(*
Nazwa:			FB_Robot2Bottles
Opis:			Robot podwójny
Wersja:			v0.91
Data:			2025-09-04
Autor:			TW,DP
Urzadzenia:		Mistsubishi
Konfiguracja:	
Zmiany:
- 20250904 [DP] EventLog-do sprawdzenia, 1 spr->wywołać błędy 
- 20241129 [DP] ReadyPlace w aborted, bRunProgramRC Aborted->Manual
Info: 

*)
FUNCTION_BLOCK FB_Robot2Bottles
VAR_INPUT
	bEnable									: BOOL;
	bRun									: BOOL;
	bPlace									: BOOL;
	bEStop									: BOOL;
	bHoming									: BOOL;
	bReset									: BOOL;
	iPickNumber								: INT;
	iPlaceNumber							: INT;
	bInkJetEnable							: BOOL;
	bPickOnlyOne							: BOOL; {warning 'Dorobić opcje pobierania tylko jednego opakowania, jeżeli będzie taka potrzeba'}
	iSpeed									: INT;
	iPickOffsetX							: INT;
	iPickOffsetY							: INT;  
	iPickOffsetZ							: INT; 
	iPick2OffsetX							: INT;
	iPick2OffsetY							: INT;  
	iPick2OffsetZ							: INT; 
	iPlace1OffsetX							: INT;
	iPlace1OffsetY							: INT;  
	iPlace1OffsetZ							: INT;
	iPlace2OffsetX							: INT;
	iPlace2OffsetY							: INT;
	iPlace2OffsetZ							: INT; 
	bEditOffset								: BOOL;		
	bManualMovement							: BOOL;
	iStationIndex							: UDINT;					
	sStationName							: STRING;		
	aDataRobotIOIn							: ARRAY[1..8] OF USINT;
	aDataRobotREGIn							: ARRAY[1..32] OF UINT;
	
	iCaseReset								: INT;
	
	iAxisId									: INT;	
	bBatteryReplacementWasMade				: BOOL;
	bGreaseReplacementWasMade				: BOOL;
	bBeltReplacementWasMade					: BOOL;
	bWarningAcknowledge						: BOOL;




END_VAR

VAR_OUTPUT
	
	eState									: E_Station;						//Stan ogólny bloku
	eRunningState							: E_RobotMovState;					//Stan podbloku
	bError									: BOOL;								//Błąd stacji
	udiErrorId								: UDINT;							//Nr błędu grzałki zasadniczej
	sErrorDescription1						: STRING(200);							//Opis błędu
	sErrorDescription2						: STRING(200);							//Opis błędu
	sErrorStationName						: STRING;							//Nazwa stacji
	udiStationID							: UDINT;							// Nr stacji

	tCycleTime								: TIME;	
	bHomingDone								: BOOL;								//Bazowanie wykonane
	bHomingNeeded 							: BOOL;								
	bCycleDone								: BOOL;
	bCycleNotDone							: BOOL;
	iLastPickNumber							: INT;
	iBottleTransferLock						: INT;
	aActualPosition							: ARRAY[0..3] OF INT;
	aLoadAxis								: ARRAY[0..3] OF INT;
	aDataRobotIOOut							: ARRAY[1..8] OF USINT;
	aDataRobotREGOut						: ARRAY[1..32] OF UINT;
	bWarning								: BOOL;
	sWarningDescription1					: STRING;
	sWarningDescription2					: STRING;
	udiWarningId							: UDINT;
	
	
END_VAR

VAR_IN_OUT
	
	bManualPick								: BOOL;
	bManualPick2							: BOOL;
	bManualPlace1							: BOOL;
	bManualPlace2							: BOOL;
	bManualReadyPosition					: BOOL;
	bManualStartInkJetPosition				: BOOL;
	bManualStopInkJetPosition				: BOOL;
	bManualWeightPosition					: BOOL;
	bManualCatch							: BOOL;
	nLubricationCounter						: DINT;	//Licznik czasu samrowania
END_VAR

VAR
	iCaseRC									: INT;
	iLastCaseRC								: INT;
	iActualCase								: INT;	
	iCaseInit								: INT;
	iCaseHoming								: INT;
	iCaseManual								: INT;
	iTemperatureRC							: INT;
	bReadyRC								: BOOL;
	bSafePositionRC							: BOOL;
	bResetErrorRC							: BOOL;
	bErrorRCActive							: BOOL;
	bServoONRC								: BOOL;
	bServoONRCActive						: BOOL;
	bServoOFFRC								: BOOL;
	bServoOFFRCActive						: BOOL;
	bOperationEnableRC						: BOOL;
	bOperationEnableRCActive				: BOOL;
	bErrorNumberRequest						: BOOL;
	bRunProgramRC							: BOOL;
	bRunProgramRCActive						: BOOL;
	bProgramResetRC							: BOOL;
	bProgramSelectRCActive					: BOOL;
	bCatcherCloseSensor						: BOOL;
	bComingUp								: BOOL;
	bSlowMotion								: BOOL;
	IODATA									: UDINT;
	ftCapFeederRobotEditOffset				: F_TRIG;
	rtCapFeederRobotEditOffset				: R_TRIG;
	tonRetryInit							: TON;	
	tonErrorDelay							: TON;	
	tonReadyError							: TON;
	iErrorCase								: INT;
	iSpeedSend								: INT;

	tonWaitForSuckerSensor					: TON;
	iZ										: INT;
	rtPick									: R_TRIG;
	
	iActualLastCase							: INT;
	aDataRobotIn							: INT;
	rtrigCycleTimerRead						: R_TRIG;
	tonCycleTimer							: TON;
	bLowLevelErrorRCActive					: BOOL;
	bWarningRCActive						: BOOL;
	bBatteryLowVoltage						: BOOL;
	bBatteryReplenishmentFinished			: BOOL;
	bGreaseReplenishmentFinished			: BOOL;
	bBeltReplenishmentFinished				: BOOL;
	tonbStateError							: TON;
	bStateError								: BOOL;
	udiHighLevelErrorId						: UDINT;
	udiMaintenanceErrorId					: UDINT;
	udiLowLevelErrorId						: UDINT;
	rtPlace									: R_TRIG;
	bHighLevelErrorRCActive					: BOOL;
	bErrorNumberRequestActive				: BOOL;
	
	fbIntTo2Byte							: FB_IntTo2Byte;
	IODATATest								: UDINT;
// dane wysyłane liczbowo do robota	
	udiIoDATARCWrite						: UDINT;	
	
	
// Wymiana smaru i paskow	
// Sygnaly wystawiane do robota
	bBatteryReplacementDone			: BOOL;	
	bGreaseReplacementDone			: BOOL;	
	bBeltReplacementDone			: BOOL;	

	
	bBeltReplacementDoneAxis3		: BOOL;
	bBeltReplacementDoneAxis4		: BOOL;
	
	bGreaseReplacementDoneAxis1		: BOOL;	
	bGreaseReplacementDoneAxis2		: BOOL;	
	bGreaseReplacementDoneAxis3		: BOOL;	
	
	
	udiErrorIdInit: UDINT;
	bWarningNumberRequest: BOOL;

	bResetWarningRC: BOOL;
	
	
		//Zmienne od EVENTLOGGER
	bAlarmInit 						: BOOL := TRUE; 
	nAlarmNumerator					: INT;
	arfbAlarm						: ARRAY[0..19] OF  FB_TcAlarm;		//Tablica bloczków błędów
	fbSourceInfo 					: FB_TcSourceInfo;
	iSourceInfo						: I_TcSourceInfo;
	sAlarmTest						: STRING;
	//Koniec zmiennych od EVENTLOGGER
END_VAR


Control();
DataExchange();
ErrorHandling();
Warning();
LubricationCounter();
aStatistic();
aStationID();

//Zabezpieczneie przed błędem 0 dp
IF udiErrorId = 0 AND bError THEN
	udiErrorId := 311;
	//udiErrorId := 999;	
END_IF

ACTION aStationID:
udiStationID	:=	iStationIndex;
END_ACTION

ACTION aStatistic:

//Statystyka do zliczania czasu cyklu 
rtrigCycleTimerRead(CLK:=bCycleDone);


	IF rtrigCycleTimerRead.Q THEN
		tCycleTime:=tonCycleTimer.ET;
	END_IF
	
tonCycleTimer(IN:= eRunningState<>E_RobotMovState.eReadyPlace , PT:=T#1D);
END_ACTION

ACTION Control:

	iSpeedSend := iSpeed;
	
	IF iPlaceNumber = 2 THEN
		iSpeedSend := REAL_TO_INT(iSpeed / 2);
	END_IF
	
	(*****Wyłączenie enable*****)
	IF NOT bEnable THEN
		IF eState <> E_Station.eDisabled AND eState <> E_Station.ePreparingToDisable THEN
				eState 				:= E_Station.ePreparingToDisable; 
		END_IF	
	END_IF

	(*****Estop*****)
	IF NOT bEstop  THEN	
		IF eState <> E_Station.eAborted AND eState <> E_Station.eAborting AND eState <> E_Station.eDisabled THEN
				eState 				:= E_Station.eAborting; 
		END_IF
	END_IF

	
	CASE eState OF
	/////////////////////////////	
		E_Station.eDisabled: 					// Stan nieaktywnosci (Stacja wyłączona) 
		
			iCaseInit				:= 0;
			IF bEnable THEN
				eState 				:= E_Station.ePreparingToReady; 
			END_IF 
			
    /////////////////////////////	    
		E_Station.eAborted: 					// Stan bezpiecznego zatrzymania (po Abortingu) 
			
			bServoONRC							:= FALSE;
			bRunProgramRC						:= FALSE;
			bResetErrorRC						:= FALSE;		
			IF bEStop THEN
				eState 				:= E_Station.ePreparingToReady;
				iCaseInit			:=0;
				eRunningState		:=	E_RobotMovState.eReadyPlace;	
			//iActualCase			:= iActualLastCase;
				//IF iActualLastCase = 200 THEN
				//	iActualCase := 250;
				//END_IF
			END_IF
			
	/////////////////////////////	
		E_Station.eAborting:                 	// Stan bezpiecznego zatrzymywania (po EStopie)
			eState 					:=	E_Station.eAborted;  
			iActualLastCase			:=	iActualCase;
		
			
	/////////////////////////////			
		E_Station.eError:                 	 	// Stan błędu 	
	
			iCaseInit				:= 0;
			//bServoONRC			:= FALSE;
			bManualPick			:= FALSE;
			bManualPick2			:= FALSE;
			bManualPlace1				:= FALSE;
			bManualPlace2					:= FALSE;
			
			IF bReset THEN
				eState 				:= E_Station.eResetting;
			END_IF
			
			IF NOT bError THEN
				eState 				:=	E_Station.ePreparingToReady;
				iCaseInit			:=0;
			END_IF
			
	/////////////////////////////
		E_Station.eResetting:					// Stan resetowania bledu (po Errorze)
			
			IF bError THEN
				
				bResetErrorRC					:= bReset;
				eRunningState					:= E_RobotMovState.eReadyPlace;
				bHomingDone						:= FALSE;
				udiErrorId						:= 0;
			END_IF
				
			IF NOT bErrorRCActive  THEN
				bError							:= FALSE;
				bResetErrorRC					:= FALSE;
				bErrorNumberRequest				:= FALSE;				
			END_IF
			
			IF NOT bError THEN
				udiErrorId 			:=	0;
   				sErrorDescription1 	:=	'';
   				sErrorDescription2 	:=	'';				
				eState 				:=	E_Station.ePreparingToReady;
				eRunningState		:=	E_RobotMovState.eReadyPlace;
				iCaseInit			:=0;
//			ELSE
//				eState 				:=	E_Station.eError;
			END_IF
        
	/////////////////////////////
		E_Station.eManualMovement:     			// Stan ruchów manualnych  
       
			ManualMovements();
			//Wyjście z trybu serwisowego
			IF NOT bManualMovement THEN
				eState:=E_Station.eReady;
			END_IF
			IF bHoming THEN
				iCaseHoming					:= 0;
				eState 						:= E_Station.eHoming; 
			END_IF

	/////////////////////////////
		E_Station.eHoming:						// Stan bazowania 
	
			Homing();
			IF NOT bHoming THEN
			   eState:=E_Station.ePreparingToReady;
			   iCaseInit			:=0;
			END_IF		
			
	/////////////////////////////
		E_Station.eHomingDone:                  // Stan wykonania bazowania 
		
			iZ:=iZ+1;
			IF NOT bHoming THEN
			   eState:=E_Station.eReady;
			END_IF
			
	/////////////////////////////
		E_Station.ePreparingToReady:            // Stan przygotowywania do gotowosci (zawsze przed Ready)  
			iCaseRC								:= 0;
			Init();
			
			
	/////////////////////////////
		E_Station.ePreparingToDisable:          // Stan przygotowywania do nieaktywnosci (po wyłączeniu Enable) 
  	
				eState:=E_Station.eDisabled;
			
	/////////////////////////////
		E_Station.eReady:						// Stan gotowosci 
		
			bServoONRC							:= TRUE;
			
			IF bServoONRCActive THEN
				bRunProgramRC					:= TRUE;			
			END_IF
		
			IF bRun AND NOT bCycleDone AND NOT bCycleNotDone THEN
				eState 						:= E_Station.eStarting; 
			END_IF
			
			
			IF bManualMovement AND bRunProgramRC THEN
				//Jeśli przejście w tryb ruchów manualnych przepisz wszystkie stany siłowników sterowanych przez moduł
				//aby zapobiec ewentualnym kolizjom po wejściu w tryb serwisowy
				iCaseManual					:= 0;
				eState 						:= E_Station.eManualMovement; 
			END_IF
			
			IF NOT bRun THEN
				bCycleDone 					:= FALSE;
				bCycleNotDone 				:= FALSE;			
			END_IF
			
			
			IF bHoming THEN
				iCaseHoming					:= 0;
				eState 						:= E_Station.eHoming; 
			END_IF
			
			
			iCaseRC							:= 0;			//22.07.2020
			
			//eRunningState					:=	E_RobotMovState.eReadyPlace;
			
			
		
			
	/////////////////////////////
		E_Station.eStopping:					// Stan zatrzymywania 

			eState 							:= E_Station.eReady;	
			
	/////////////////////////////
		E_Station.eStarting:                  	// Stan uruchamiania (po Ready)	
			bResetErrorRC					:= FALSE;	
			eState					 		:= E_Station.eRunning; 
			
	/////////////////////////////
		E_Station.eRunning:               		// Stan wykonywania cyklu (po Startingu), w tym stanie osobny
 

			IF NOT bRun AND NOT bCycleDone THEN					(*Przerywanie cyklu*)
				eState 				 		:= E_Station.eStopping;	
			END_IF
			
			IF bCycleDone OR bCycleNotDone THEN (*Cykl zakończony*)
				eState 				 		:= E_Station.eReady;
				eRunningState						:=	E_RobotMovState.eReadyPlace;
			END_IF		
			
			Running();
			
			
	/////////////////////////////		
	END_CASE
END_ACTION

ACTION DataExchange:


//SignalOutput
aDataRobotIOOut[1].0                	:= bOperationEnableRC;
aDataRobotIOOut[1].1                	:= bRunProgramRC;
aDataRobotIOOut[1].2              		:= bSlowMotion;
aDataRobotIOOut[1].3                	:= bProgramResetRC;
aDataRobotIOOut[1].4                	:= bServoONRC;
aDataRobotIOOut[1].5                	:= bServoOFFRC;
aDataRobotIOOut[1].6                	:= bResetErrorRC OR bResetWarningRC;
aDataRobotIOOut[1].7                	:= bEditOffset;
aDataRobotIOOut[2].0                	:= bManualCatch;
aDataRobotIOOut[2].1                	:= bErrorNumberRequest OR bWarningNumberRequest;
//Dodane Darek
aDataRobotIOOut[2].7                	:= bBatteryReplacementDone;		//6015
aDataRobotIOOut[3].0                	:= bGreaseReplacementDone;		//6016
aDataRobotIOOut[3].1                	:= bBeltReplacementDone;		//6017
aDataRobotIOOut[3].2                	:= bBeltReplacementDone;		//6017

//SignalRegOutput
aDataRobotREGOut[1]                    	:= INT_TO_UINT(iCaseRC);
aDataRobotREGOut[2]                    	:= INT_TO_UINT(iSpeedSend);
aDataRobotREGOut[3]                    	:= INT_TO_UINT(iPickOffsetX);
aDataRobotREGOut[4]                    	:= INT_TO_UINT(iPickOffsetY);
aDataRobotREGOut[5]                    	:= INT_TO_UINT(iPickOffsetZ);
aDataRobotREGOut[6]                    	:= INT_TO_UINT(iPlace1OffsetX);
aDataRobotREGOut[7]                  	:= INT_TO_UINT(iPlace1OffsetY);
aDataRobotREGOut[8]                    	:= INT_TO_UINT(iPlace1OffsetZ);
aDataRobotREGOut[9]                    	:= INT_TO_UINT(iPlace2OffsetX);
aDataRobotREGOut[10]                	:= INT_TO_UINT(iPlace2OffsetY);
aDataRobotREGOut[11]                	:= INT_TO_UINT(iPlace2OffsetZ);
//Dodane Darek
aDataRobotREGOut[12]                    := INT_TO_UINT(iPick2OffsetX);
aDataRobotREGOut[13]                    := INT_TO_UINT(iPick2OffsetY);
aDataRobotREGOut[14]                    := INT_TO_UINT(iPick2OffsetZ);

// IODATA

fbIntTo2Byte(
iInput:= UDINT_TO_INT(udiIoDATARCWrite), 
byStarszy=> , 
byMlodszy=> );


aDataRobotIOOut[8]												:= fbIntTo2Byte.byStarszy;
aDataRobotIOOut[7]												:= fbIntTo2Byte.byMlodszy;

// Testowy odczyt wartosci wysyłanej
IODATATest                                	:= WORD_TO_UDINT(F_2Bytes_To_Word(aDataRobotIOOut[8], aDataRobotIOOut[7]));


//SignalInput                               
bOperationEnableRCActive            	:= aDataRobotIOIn[1].0;		//6000
bRunProgramRCActive                   	:= aDataRobotIOIn[1].1;
//                                    	:= aDataRobotIOIn[1].2;
bProgramSelectRCActive                	:= aDataRobotIOIn[1].3;
bServoONRCActive                    	:= aDataRobotIOIn[1].4;
bServoOFFRCActive                    	:= aDataRobotIOIn[1].5;
bErrorRCActive                        	:= aDataRobotIOIn[1].6;
bReadyRC                            	:= aDataRobotIOIn[1].7;
bSafePositionRC                        	:= aDataRobotIOIn[2].0;		//6008
bErrorNumberRequestActive               := aDataRobotIOIn[2].1;
bCatcherCloseSensor                    	:= aDataRobotIOIn[2].2;

//Dodane Darek
bHighLevelErrorRCActive                 := aDataRobotIOIn[2].3;		//6011
bLowLevelErrorRCActive                  := aDataRobotIOIn[2].4;		//6012
bWarningRCActive                    	:= aDataRobotIOIn[2].5;		//6013
bBatteryLowVoltage              		:= aDataRobotIOIn[2].6;		//6014
bBatteryReplenishmentFinished               := aDataRobotIOIn[2].7;		//6015
bGreaseReplenishmentFinished	            := aDataRobotIOIn[3].0;		//6016
bBeltReplenishmentFinished	                := aDataRobotIOIn[3].1;		//6017



//SignalRegInput
iActualCase                            	:= UINT_TO_INT(aDataRobotREGIn[1]);
aLoadAxis[0]                        	:= UINT_TO_INT(aDataRobotREGIn[2]);
aLoadAxis[1]                        	:= UINT_TO_INT(aDataRobotREGIn[3]);       
aLoadAxis[2]                        	:= UINT_TO_INT(aDataRobotREGIn[4]);       
aLoadAxis[3]                        	:= UINT_TO_INT(aDataRobotREGIn[5]);
IODATA                                	:= WORD_TO_UDINT(F_2Bytes_To_Word(aDataRobotIOIn[8], aDataRobotIOIn[7]));
END_ACTION

ACTION ErrorDescription:
IF bErrorRCActive AND bHighLevelErrorRCActive THEN

		CASE udiHighLevelErrorId OF	
			
			
0001:					
					
	sErrorDescription1 := 'Fail safe error (SRVOFF).  System problem.';				
	sErrorDescription2 := 'Turn the power OFF and ON once. When it comes back, contact to the dealer.';				
					
0002:					
					
	sErrorDescription1 := 'Fail safe error (STOP).  System Problem.';				
	sErrorDescription2 := 'Turn the power OFF and ON once. When it comes back, contact to the dealer.';				
					
0003:					
					
	sErrorDescription1 := 'System fail.  System Problem.';				
	sErrorDescription2 := 'Check System.When it comes back, contact to the dealer.';				
					
0004:					
					
	sErrorDescription1 := 'CPU Watch dog error.  CPU was not normally treatable.';				
	sErrorDescription2 := 'It is necessary to change some parts when not improvement';				
					
0005:					
					
	sErrorDescription1 := 'Turn the power OFF and ON onc.  The robot model was selected..';				
	sErrorDescription2 := 'Turn the power OFF and ON once';				
					
0006:					
					
	sErrorDescription1 := ' CPU process error.  CPU was not normally treatable.';				
	sErrorDescription2 := 'It is necessary to change some parts when not improvement';				
					
0008:					
					
	sErrorDescription1 := ' CPU synchronization error.  CPU synchronization was failed.';				
	sErrorDescription2 := 'Turn the power OFF and ON once';				
					
0009:					
					
	sErrorDescription1 := 'Version UP (ALL).  Version UP (ALL).';				
	sErrorDescription2 := 'Turn the power OFF,ROTSW=0 and power ON once';				
					
0010:					
					
	sErrorDescription1 := 'Illeagal Version (file).  Version is different.';				
	sErrorDescription2 := 'File was initialized';				
					
0011:					
					
	sErrorDescription1 := 'Illeagal Version (system data.  Version is different.';				
	sErrorDescription2 := 'System data was initialized';				
					
0012:					
					
	sErrorDescription1 := 'Initialize (error log).  Version is different or illegal log file.';				
	sErrorDescription2 := 'Error log was initialized';				
					
0014:					
					
	sErrorDescription1 := 'System error (illegal MECHA).  System error (illegal MECHA).';				
	sErrorDescription2 := 'Set the correct MECHA';				
					
0015:					
					
	sErrorDescription1 := 'Illeagal Version (file).  System ERROR 1.';				
	sErrorDescription2 := 'Contact the maker.';				
					
0016:					
					
	sErrorDescription1 := 'Turn the power OFF and ON onc.  Power OFF/ON a little more slowly,please.';				
	sErrorDescription2 := 'Turn the power OFF and ON once';				
					
0017:					
					
	sErrorDescription1 := '  EEPROM error.  EEPROM is broken.';				
	sErrorDescription2 := 'It is necessary to replace the CPU board';				
					
0019:					
					
	sErrorDescription1 := 'Illegal RotSW on CPU.  RotSW is set not 0.';				
	sErrorDescription2 := 'Please set RotSW to 0';				
					
0020:					
					
	sErrorDescription1 := 'System Error(same name is Bac.  System Error(same name is Backup data.).';				
	sErrorDescription2 := 'Change the system software';				
					
0021:					
					
	sErrorDescription1 := 'System Error(Backup data is C.  System Error(Backup data is Count over.).';				
	sErrorDescription2 := 'Change the system software';				
					
0022:					
					
	sErrorDescription1 := 'System Error(Backup data is n.  System Error(Backup data is no area.).';				
	sErrorDescription2 := 'Change the system software';				
					
0025:					
					
	sErrorDescription1 := ' Files will be saved to ROM.  Program and parameter files will be saved to ROM.';				
	sErrorDescription2 := 'Turn the power OFF and power ON once';				
					
0026:					
					
	sErrorDescription1 := ' Files will be loaded from ROM.  Program and parameter files will be loaded from ROM.';				
	sErrorDescription2 := 'Turn the power OFF and power ON once';				
					
0027:					
					
	sErrorDescription1 := ' Backup or restore is canceled.  Backup or restore is canceled.';				
	sErrorDescription2 := 'Turn the power OFF and power ON once';				
					
0028:					
					
	sErrorDescription1 := ' Memory error (ECC).  2bit error of ECC was detected.';				
	sErrorDescription2 := 'Turn the power OFF and ON once';				
					
0039:					
					
	sErrorDescription1 := 'Door Switch Signal line is fa.  Door Switch Signal line is faulty..';				
	sErrorDescription2 := 'Check the Door Switch Signal line';				
					
0040:					
					
	sErrorDescription1 := 'Door Switch Signal is Input.  Door Switch is opened.';				
	sErrorDescription2 := 'Please close the Door be connected with Door Switch';				
					
0041:					
					
	sErrorDescription1 := 'Comm. error (Remote I/O #1).  Communication line is illegal.';				
	sErrorDescription2 := 'Check the cable or power supply';				
					
0042:					
					
	sErrorDescription1 := ' Comm. error (Remote I/O #2).  Communication line is illegal.';				
	sErrorDescription2 := 'Check the cable or power supply';				
					
0043:					
					
	sErrorDescription1 := ' Comm. error (Remote I/O #3).  Communication line is illegal.';				
	sErrorDescription2 := 'Check the cable or power supply';				
					
0044:					
					
	sErrorDescription1 := ' Comm. error (Remote I/O #4).  Communication line is illegal.';				
	sErrorDescription2 := 'Check the cable or power supply';				
					
0045:					
					
	sErrorDescription1 := ' Comm. error (Remote I/O #5).  Communication line is illegal.';				
	sErrorDescription2 := 'Check the cable or power supply';				
					
0046:					
					
	sErrorDescription1 := ' Faulty wiring (Mode sel. swit.  The state of doubled wiring is not matching (Mode sel. switch).';				
	sErrorDescription2 := 'Please check the wiring (Mode sel. switch)';				
					
0047:					
					
	sErrorDescription1 := ' OCL detect.  OCL detect.';				
	sErrorDescription2 := 'Please check the line (O/P Emergency Stop)';				
					
0048:					
					
	sErrorDescription1 := ' Faulty line (Mode Selector SW.  The state of doubled line is not matching (Mode Selector switch).';				
	sErrorDescription2 := 'Please check the line (Mode Selector switch)';				
					
0049:					
					
	sErrorDescription1 := ' Faulty Line (T/B Enable Switc.  The state of doubled line is not matching (T/B Enable Switch).';				
	sErrorDescription2 := 'Please check the line (T/B Enable Switch)';				
					
0050:					
					
	sErrorDescription1 := 'EMG signal is input. (externa.  EMG signal is input. (external).';				
	sErrorDescription2 := 'Check the external emergency stop';				
					
0051:					
					
	sErrorDescription1 := 'EMG line is faulty.(external).  EMG line is faulty.(external).';				
	sErrorDescription2 := 'Check the external emergency stop';				
					
0052:					
					
	sErrorDescription1 := ' EMG signal is input.(Add.Axis.  EMG signal is input.(Add.Axis1).';				
	sErrorDescription2 := 'Check the emergency stop of Additional Axis card';				
					
0053:					
					
	sErrorDescription1 := 'EMG signal is input.(Add.Axis.  EMG signal is input.(Add.Axis).';				
	sErrorDescription2 := 'Check the emergency stop of Additional Axis servo amp.';				
					
0054:					
					
	sErrorDescription1 := ' Faulty wiring (External EMG p.  The state of doubled wiring is not matching (External EMG).';				
	sErrorDescription2 := 'Please check the wiring (External Emergency Stop)';				
					
0060:					
					
	sErrorDescription1 := 'EMG signal is input. (O.Panel.  EMG signal is input. (O.Panel).';				
	sErrorDescription2 := 'Check the O.Panel emergency stop';				
					
0061:					
					
	sErrorDescription1 := 'EMG line is faulty.(0.Panel).  EMG line is faulty.(0.Panel).';				
	sErrorDescription2 := 'Check the O.Panel emergency stop';				
					
0070:					
					
	sErrorDescription1 := 'EMG signal is input. (T.Box).  EMG signal is input. (T.Box).';				
	sErrorDescription2 := 'Check the T.Box emergency stop';				
					
0071:					
					
	sErrorDescription1 := 'EMG line is faulty.(T.Box).  EMG line is faulty.(T.Box).';				
	sErrorDescription2 := 'Check the T.Box emergency stop';				
					
0072:					
					
	sErrorDescription1 := 'EMG cancel operation is fault.  TB cancel switch operation was incorrect.';				
	sErrorDescription2 := 'Check the T/B cancel switch operation';				
					
0073:					
					
	sErrorDescription1 := 'EMG cancel line is faulty.(T..  EMG cancel line is faulty.(T.Box).';				
	sErrorDescription2 := 'Check the EMG cancel line';				
					
0074:					
					
	sErrorDescription1 := 'Faulty line (T/B Enable/Disab.  The state of doubled line is not matching (T/B Enable/Disable).';				
	sErrorDescription2 := 'Please check the line (T/B Enable/Disable)';				
					
0075:					
					
	sErrorDescription1 := 'TB communication error.  Communication between the RC and TB was cut off.';				
	sErrorDescription2 := 'Check TB communication line';				
					
0076:					
					
	sErrorDescription1 := 'TB connection error.  Cannot detect TB connection.';				
	sErrorDescription2 := 'If this error recurs, please contact us';				
					
0077:					
					
	sErrorDescription1 := ' Electric double layer overvol.  A power supply of a substrate in the robot is broken.';				
	sErrorDescription2 := 'Turn the power OFF and contact your service provider';				
					
0079:					
					
	sErrorDescription1 := ' Contactor of converter unit e.  Contactor of converter unit is closed.';				
	sErrorDescription2 := 'Confirm status of contactor of converter unit';				
					
0080:					
					
	sErrorDescription1 := ' Fuse of brake line is blown.  Fuse of brake line is blown.';				
	sErrorDescription2 := 'Change fuse';				
					
0081:					
					
	sErrorDescription1 := ' Fuse is blown.(motor hand I/F.  Fuse is blown.(motor hand I/F).';				
	sErrorDescription2 := 'Change fuse';				
					
0082:					
					
	sErrorDescription1 := 'Fuse is broken (air hand I/F).  Fuse is blown.(air hand I/F).';				
	sErrorDescription2 := 'Change fuse';				
					
0083:					
					
	sErrorDescription1 := 'Fuse is broken(hand input pow.  Fuse is blown.(hand input power).';				
	sErrorDescription2 := 'Change fuse';				
					
0084:					
					
	sErrorDescription1 := 'Fuse is broken(O/P).  Fuse is blown.(O/P).';				
	sErrorDescription2 := 'Change fuse';				
					
0085:					
					
	sErrorDescription1 := ' Fuse is blown.(External EMG).  Open phase in the input power.';				
	sErrorDescription2 := 'Change fuse';				
					
0086:					
					
	sErrorDescription1 := 'Hand module overcurrent.  Hand module is broken.';				
	sErrorDescription2 := 'Change Hand module';				
					
0087:					
					
	sErrorDescription1 := 'Fuse is blown.(Brake).  Fuse is blown.(Brake).';				
	sErrorDescription2 := 'Change fuse';				
					
0088:					
					
	sErrorDescription1 := ' Fuse is blown.(Service I/F).  Fuse is blown.(Service I/F).';				
	sErrorDescription2 := 'Please confirm the input and output current of service I/F. ';				
					
0089:					
					
	sErrorDescription1 := ' Fuse of external battery is b.  Fuse of external battery is blown..';				
	sErrorDescription2 := 'Check that an outside power-supply voltage is 4.5V or less.';				
					
0090:					
					
	sErrorDescription1 := ' Fuse is blown..  Fuse is blown.';				
	sErrorDescription2 := 'Change fuse';				
					
0093:					
					
	sErrorDescription1 := ' Safety relay fuse is blown..  Safety relay fuse is blown..';				
	sErrorDescription2 := 'Change fuse.';				
					
0094:					
					
	sErrorDescription1 := ' The fuse in the T/B was blown.  The fuse in the T/B power supply line was blown..';				
	sErrorDescription2 := 'Please check the earth fault of the T/B cable.';				
					
0097:					
					
	sErrorDescription1 := ' Faulty status (MC).  The state of doubled signal is not matching (MC status).';				
	sErrorDescription2 := 'Turn the power OFF and ON once';				
					
0098:					
					
	sErrorDescription1 := ' Faulty status (SR).  The state of doubled signal is not matching (SR status).';				
	sErrorDescription2 := 'Turn the power OFF and ON once';				
					
0099:					
					
	sErrorDescription1 := ' S/W with an old version is in.  S/W with an old version is installed.';				
	sErrorDescription2 := 'Install the S/W with a correct version';				
					
0100:					
					
	sErrorDescription1 := 'Temperature in the Controlle .  FAN check or Filter at the bottom on Controller becomes old.';				
	sErrorDescription2 := 'Please exchange the filter to new filter or clean up the filter';				
					
0103:					
					
	sErrorDescription1 := ' Temp. in robot CPU is too hig.  Ambient temperature of robot CPU becomes high.';				
	sErrorDescription2 := 'Please lower ambient temperature to the specification range';				
					
0117:					
					
	sErrorDescription1 := ' Power supply error (brake).  The output of the power supply deviated from the specified range.';				
	sErrorDescription2 := 'Turn the power OFF and contact your service provider';				
					
0130:					
					
	sErrorDescription1 := 'System RemoteI/O down.  Communication line of System Remote I/O is illegal.';				
	sErrorDescription2 := 'Check the cable or power supply';				
					
0131:					
					
	sErrorDescription1 := ' Plural Ope-panel are installe.  One operation panel can be installed..';				
	sErrorDescription2 := 'Install only one operation panel.';				
					
0140:					
					
	sErrorDescription1 := 'Fuse is blown.(Safety unit).  Fuse is blown.(Safety unit).';				
	sErrorDescription2 := 'Change fuse';				
					
0141:					
					
	sErrorDescription1 := ' Wiring error of EMGIN connect.  Wiring error of EMGIN connector.';				
	sErrorDescription2 := 'Please confirm the wiring for EMGIN';				
					
0160:					
					
	sErrorDescription1 := 'Cannot use PIO I/F and Unit.  The I/O Channel number of PIO interface and PIO unit overlaps..';				
	sErrorDescription2 := 'Select either of Paralle I/O interface or Paralle I/O unit.';				
					
0162:					
					
	sErrorDescription1 := 'Cannot use PIO I/F and Unit.  The I/O Channel number of PIO interface and PIO unit overlaps..';				
	sErrorDescription2 := 'Select either of Paralle I/O interface or Paralle I/O unit.';				
					
0163:					
					
	sErrorDescription1 := 'Cannot use PIO I/F and Unit.  The I/O Channel number of PIO interface and PIO unit overlaps..';				
	sErrorDescription2 := 'Select either of Paralle I/O interface or Paralle I/O unit.';				
					
0170:					
					
	sErrorDescription1 := 'Parallel I/O interface H/W er.  The card might be broken..';				
	sErrorDescription2 := 'Please exchange the Parallel I/O interface card.';				
					
0172:					
					
	sErrorDescription1 := 'Parallel I/O interface H/W er.  The card might be broken..';				
	sErrorDescription2 := 'Please exchange the Parallel I/O interface card.';				
					
0173:					
					
	sErrorDescription1 := 'Parallel I/O interface H/W er.  The card might be broken..';				
	sErrorDescription2 := 'Please exchange the Parallel I/O interface card.';				
					
0180:					
					
	sErrorDescription1 := 'Fuse is blown.(PIO) （Slot 1-F.  Fuse is blown.(Paralle I/O interface).';				
	sErrorDescription2 := 'Change fuse (Paralle I/O interface)';				
					
0182:					
					
	sErrorDescription1 := 'Fuse is blown.(PIO) （Slot 2-F.  Fuse is blown.(Paralle I/O interface).';				
	sErrorDescription2 := 'Change fuse (Paralle I/O interface)';				
					
0183:					
					
	sErrorDescription1 := 'Fuse is blown.(PIO) （Slot 3-F.  Fuse is blown.(Paralle I/O interface).';				
	sErrorDescription2 := 'Change fuse (Paralle I/O interface)';				
					
0210:					
					
	sErrorDescription1 := ' Power supply error.  The output of the power supply deviated from the specified range.';				
	sErrorDescription2 := 'Turn the power OFF and ON once';				
					
0211:					
					
	sErrorDescription1 := ' Power supply error.  The output of the power supply deviated from the specified range.';				
	sErrorDescription2 := 'Turn the power OFF and ON once';				
					
0212:					
					
	sErrorDescription1 := ' Power supply error.  The output of the power supply deviated from the specified range.';				
	sErrorDescription2 := 'Turn the power OFF and ON once';				
					
0213:					
					
	sErrorDescription1 := ' Power supply error.  The output of the power supply deviated from the specified range.';				
	sErrorDescription2 := 'Turn the power OFF and ON once';				
					
0220:					
					
	sErrorDescription1 := ' Memory error (Main CPU).  Memory error was detected (Main CPU).';				
	sErrorDescription2 := 'Turn the power OFF and ON once';				
					
0230:					
					
	sErrorDescription1 := ' Safety parameter error.  Detect errors in safety parameter value.';				
	sErrorDescription2 := 'Please check the safety parameter setting';				
					
0231:					
					
	sErrorDescription1 := ' Parameter CRC error.  Detect CRC errors in safety parameter.';				
	sErrorDescription2 := 'Please check the safety parameters settings and write parameters';				
					
0241:					
					
	sErrorDescription1 := ' Fault in Safety Communication.  Detect a fault in safety communication.';				
	sErrorDescription2 := 'Turn the power OFF and ON once';				
					
0242:					
					
	sErrorDescription1 := ' Fault in Safety Data.  Detect a fault in safety data.';				
	sErrorDescription2 := 'Turn the power OFF and ON once';				
					
0243:					
					
	sErrorDescription1 := ' Safety function unavailable.  The Safety Function is not supported by this robot.';				
	sErrorDescription2 := 'Disable the safety function';				
					
0260:					
					
	sErrorDescription1 := ' EMG circuit diagnosis error.  Voltage diagnosis error.';				
	sErrorDescription2 := 'Turn the power OFF and ON once';				
					
0270:					
					
	sErrorDescription1 := ' Voltage diagnosis error.  Voltage diagnosis error.';				
	sErrorDescription2 := 'Turn the power OFF and ON once';				
					
0280:					
					
	sErrorDescription1 := ' STO circuit diagnosis error.  STO citcuit error.';				
	sErrorDescription2 := 'Turn the power OFF and ON once';				
					
0290:					
					
	sErrorDescription1 := ' PLD control error.  PLD control error.';				
	sErrorDescription2 := 'Turn the power OFF and ON once';				
					
0300:					
					
	sErrorDescription1 := ' CR800 test H-Error.  General-purpose H-Error for the function test of CR800.';				
	sErrorDescription2 := 'Check the embedded message';				
					
0310:					
					
	sErrorDescription1 := ' Mecha board access error.  Failed in access to a Mecha board.';				
	sErrorDescription2 := 'Please confirm the connection with Mecha board';				
					
0311:					
					
	sErrorDescription1 := ' RemoteI/O unit config error.  The multiple RemoteI/O units which do not support are connected.';				
	sErrorDescription2 := 'Please confirm the constitution of RemoteI/O unit';				
					
0315:					
					
	sErrorDescription1 := ' Can not access the D-device are.  This area cannot be used in duplicate.';				
	sErrorDescription2 := 'Please change the D-device start number in parameter DDEVVLn';				
					
0316:					
					
	sErrorDescription1 := ' The D-device area is out of r.  An area corresponding to the variable type can not be allocated.';				
	sErrorDescription2 := 'Please change the D-device start number in parameter DDEVVLn';				
					
0317:					
					
	sErrorDescription1 := ' The D-device variable duplica.  Cannot be doubly allotted to one variable.';				
	sErrorDescription2 := 'Please change the variable name in parameter DDEVVLn';				
					
0470:					
					
	sErrorDescription1 := ' Abnormality of DB(Add.Axis).  The addition axis dynamic brake is abnormal.';				
	sErrorDescription2 := 'Check the dynamic brake unit and the cable connection';				
					
0490:					
					
	sErrorDescription1 := 'Alarm of fan in the robot.  Fan in the robot might be out of order.';				
	sErrorDescription2 := 'Please exchange the fan in the robot';				
					
0491:					
					
	sErrorDescription1 := 'Alarm of fan1 in the robot.  Fan1 in the robot might be out of order.';				
	sErrorDescription2 := 'Please exchange the fan1 in the robot';				
					
0492:					
					
	sErrorDescription1 := 'Alarm of fan2 in the robot.  Fan2 in the robot might be out of order.';				
	sErrorDescription2 := 'Please exchange the fan2 in the robot';				
					
0493:					
					
	sErrorDescription1 := 'Alarm of fan3 in the robot.  Fan3 in the robot might be out of order.';				
	sErrorDescription2 := 'Please exchange the fan3 in the robot';				
					
0494:					
					
	sErrorDescription1 := 'Alarm of fan4 in the robot.  Fan4 in the robot might be out of order.';				
	sErrorDescription2 := 'Please exchange the fan4 in the robot';				
					
0495:					
					
	sErrorDescription1 := 'Alarm of fan5 in the robot.  Fan5 in the robot might be out of order.';				
	sErrorDescription2 := 'Please exchange the fan5 in the robot';				
					
0496:					
					
	sErrorDescription1 := 'Alarm of fan6 in the robot.  Fan6 in the robot might be out of order.';				
	sErrorDescription2 := 'Please exchange the fan6 in the robot';				
					
0497:					
					
	sErrorDescription1 := 'Alarm of fan7 in the robot.  Fan7 in the robot might be out of order.';				
	sErrorDescription2 := 'Please exchange the fan7 in the robot';				
					
0498:					
					
	sErrorDescription1 := 'Alarm of fan8 in the robot.  Fan8 in the robot might be out of order.';				
	sErrorDescription2 := 'Please exchange the fan8 in the robot';				
					
0500:					
					
	sErrorDescription1 := 'Servo axis setting error.  The setting of the axis number selection switch is illegal.';				
	sErrorDescription2 := 'Confirm the setting of the axis selection switch';				
					
0510:					
					
	sErrorDescription1 := 'The converter setting is ille.  The setting of the external emergency stop mode is illegal.';				
	sErrorDescription2 := 'Correctly set';				
					
0520:					
					
	sErrorDescription1 := 'Robot axis setting illegal.  The axis No is duplicated with another robot axis No.';				
	sErrorDescription2 := 'Correctly set';				
					
0530:					
					
	sErrorDescription1 := 'Servo sys. error (memory).  The servo amplifier memory ICs check sum is illegal.';				
	sErrorDescription2 := 'Turn the power OFF and ON once';				
					
0540:					
					
	sErrorDescription1 := 'Servo sys. error (over run).  The servo amp. / motion task S/W did not end within the specified time.';				
	sErrorDescription2 := 'Turn the power OFF and ON once';				
					
0550:					
					
	sErrorDescription1 := 'Servo sys. error (mag. pole p.  the magnetic pole position signal from encoderis illegal.';				
	sErrorDescription2 := 'Turn the power OFF and ON once';				
					
0560:					
					
	sErrorDescription1 := 'Servo sys. error (A/D）.  the magnetic pole position signal from encoderis illegal.';				
	sErrorDescription2 := 'Turn the power OFF and ON once';				
					
0570:					
					
	sErrorDescription1 := 'Encoder error (EEPROM).  the magnetic pole position signal from encoderis illegal.';				
	sErrorDescription2 := 'Turn the power OFF and ON once';				
					
0580:					
					
	sErrorDescription1 := 'Encoder error (LED).  The LED of encoder has deteriorated.';				
	sErrorDescription2 := 'Turn the power OFF and ON once';				
					
0590:					
					
	sErrorDescription1 := 'Encoder error (position data).  the per rotation position data is illegal.';				
	sErrorDescription2 := 'Turn the power OFF and ON once';				
					
0600:					
					
	sErrorDescription1 := 'Encoder no-signal detection1.  An error was detected in the operation input of the encoder.';				
	sErrorDescription2 := 'Turn the power OFF and ON once';				
					
0610:					
					
	sErrorDescription1 := 'Encoder no-signal detection2.  An error was detected in the operation input of the encoder.';				
	sErrorDescription2 := 'Turn the power OFF and ON once';				
					
0620:					
					
	sErrorDescription1 := 'Servo amplifier LSI error.  An error was detected in the operation of the servo AMP LSI.';				
	sErrorDescription2 := 'Turn the power OFF and ON once';				
					
0630:					
					
	sErrorDescription1 := 'Unused axis servo error.  A power module error occurred in an axis not used.';				
	sErrorDescription2 := 'Turn the power OFF and ON once';				
					
0640:					
					
	sErrorDescription1 := 'System error (ABS CPU).  Error in the CPU of the absolute position linear scale.';				
	sErrorDescription2 := 'Turn the power OFF and ON once';				
					
0650:					
					
	sErrorDescription1 := 'Absolute position error.  Error in the circuit of the absolute position linear scale.';				
	sErrorDescription2 := 'Turn the power OFF and ON once';				
					
0660:					
					
	sErrorDescription1 := 'Incremental position error.  Error in the incremental position detection circuit.';				
	sErrorDescription2 := 'Turn the power OFF and ON once';				
					
0670:					
					
	sErrorDescription1 := 'Encoder CPU error.  An error was detected in the CPU of the encoder.';				
	sErrorDescription2 := 'Turn the power OFF and ON once';				
					
0680:					
					
	sErrorDescription1 := 'Encoder LED error.  Deterioration of the encoder LED was detected.';				
	sErrorDescription2 := 'Turn the power OFF and ON once';				
					
0690:					
					
	sErrorDescription1 := ' regeneration circuit error.  A regenerative transistor or resistor error was detected.';				
	sErrorDescription2 := 'Turn the power OFF and ON once';				
					
0700:					
					
	sErrorDescription1 := 'P.S. external contactor fusin.  The external contactor turned ON even at READY OFF.';				
	sErrorDescription2 := 'Turn the power OFF and ON once';				
					
0710:					
					
	sErrorDescription1 := 'Power supply rush relay error.  The relay on servo cpu card did not turn ON.';				
	sErrorDescription2 := 'Turn the power OFF and ON once';				
					
0711:					
					
	sErrorDescription1 := 'Power supply relay error.  The discharge relay on converter card did not turn ON.';				
	sErrorDescription2 := 'Turn the power OFF and ON once';				
					
0712:					
					
	sErrorDescription1 := ' Converter fuse fusing.  Fuse of a converter fused for a ground fault or short circuit.';				
	sErrorDescription2 := 'Please exchange a fuse of a converter';				
					
0713:					
					
	sErrorDescription1 := ' Encoder power supply fuse tri.  Encoder power supply fuse tripped by ground fault, short circuit.';				
	sErrorDescription2 := 'Turn the power OFF, wait a while, and then turn ON again';				
					
0720:					
					
	sErrorDescription1 := 'Power supply watch dog.  The power supply S/W did not end within the specified time.';				
	sErrorDescription2 := 'Turn the power OFF and ON once';				
					
0730:					
					
	sErrorDescription1 := 'Power supply rush relay fusin.  The rush resistance short-circuit relay did not turn OFF.';				
	sErrorDescription2 := 'Turn the power OFF and ON once';				
					
0740:					
					
	sErrorDescription1 := 'Power supply main circuit err.  The main circuit capacitor was not charged correctly.';				
	sErrorDescription2 := 'Turn the power OFF and ON once';				
					
0742:					
					
	sErrorDescription1 := ' Power supply main circuit err.  A main circuit voltage has decreased because of Safety relay.';				
	sErrorDescription2 := 'Check for errors in the Safety relay';				
					
0743:					
					
	sErrorDescription1 := ' Power supply main circuit err.  A main circuit voltage has decreased because of contactor fail..';				
	sErrorDescription2 := 'Check for errors in the contactor.';				
					
0750:					
					
	sErrorDescription1 := 'Power supply memory error.  An error was detected in the power supply memory circuit.';				
	sErrorDescription2 := 'Turn the power OFF and ON once';				
					
0760:					
					
	sErrorDescription1 := 'Power supply error.  An error was detected in the data comm. with the power supply.';				
	sErrorDescription2 := 'Turn the power OFF and ON once';				
					
0770:					
					
	sErrorDescription1 := 'Power supply process error.  An error occurred in the process cycle of power supply.';				
	sErrorDescription2 := 'Turn the power OFF and ON once';				
					
0780:					
					
	sErrorDescription1 := 'Servo amplifier watch dog.  The Servo amplifier S/W did not end within the specified time.';				
	sErrorDescription2 := 'Turn the power OFF and ON once';				
					
0790:					
					
	sErrorDescription1 := 'Servo amplifier boad error.  An error was detected in the servo amplifier PCB.';				
	sErrorDescription2 := 'Turn the power OFF and ON once';				
					
0800:					
					
	sErrorDescription1 := 'Servo amplifier clock error.  An error was detected in the servo amplifier clock.';				
	sErrorDescription2 := 'Turn the power OFF and ON once';				
					
0810:					
					
	sErrorDescription1 := 'Power supply undervoltage.  Insufficient bus voltage was detected in main circuit.';				
	sErrorDescription2 := 'Check the power supply connection and power supply state';				
					
0820:					
					
	sErrorDescription1 := 'Motor ground fault.  A motor cable ground fault was detected.';				
	sErrorDescription2 := 'Check the motor cables connection and conductivity';				
					
0830:					
					
	sErrorDescription1 := 'Servo amplifier overvoltage.  The main circuit bus voltage exceeded the tolerable value.';				
	sErrorDescription2 := 'Check the power voltage and regenerative resistance value';				
					
0840:					
					
	sErrorDescription1 := 'Instantaneous power failure(S.  The power was OFF for 50msec or more.';				
	sErrorDescription2 := 'Check the power supply connection and power supply state';				
					
0850:					
					
	sErrorDescription1 := 'Power supply voltage incorrec.  Open phase in the input power, or the voltage is outof range.';				
	sErrorDescription2 := 'Check the power supply connection and power supply state';				
					
0860:					
					
	sErrorDescription1 := 'Power supply overvoltage.  The main circuit bus voltage exceeded the tolerable value.';				
	sErrorDescription2 := 'Check the power supply connection and power supply state';				
					
0870:					
					
	sErrorDescription1 := 'Power module overheat (Fan St.  A cooling fan stopped, and overheat occurred.';				
	sErrorDescription2 := 'Check the rotation of fan, and the connector connected to a fan';				
					
0880:					
					
	sErrorDescription1 := 'Power module overheat.  Overheating of the power module (IPM) was detected.';				
	sErrorDescription2 := 'Turn the power OFF, wait a while, and then turn ON again';				
					
0890:					
					
	sErrorDescription1 := 'Servo amplifier motor overhea.  The motor or detectors thermal protector activated.';				
	sErrorDescription2 := 'Turn the power OFF, wait a while, and then turn ON again';				
					
0900:					
					
	sErrorDescription1 := 'Absolute position overspeed.  The absolute position linear scale moved 45mm/s or more.';				
	sErrorDescription2 := 'Turn the power OFF and ON once';				
					
0910:					
					
	sErrorDescription1 := 'Servo amplifier overspeed.  The motor speed rose to 1.2 times the rating.';				
	sErrorDescription2 := 'Turn the power OFF and ON once';				
					
0920:					
					
	sErrorDescription1 := 'Power module overcurrent.  An overcurrent was detected in the  power supply IPM.';				
	sErrorDescription2 := 'Check the motor cables connection and conductivity';				
					
0930:					
					
	sErrorDescription1 := 'Motor overcurrent.  An excessive current flowed to the motor.';				
	sErrorDescription2 := 'Turn the power OFF and ON once';				
					
0940:					
					
	sErrorDescription1 := 'Overload 1.  Run in the overload range set with SVOLL and SVOLT.';				
	sErrorDescription2 := 'Check the load weight and the robot for collisions, etc';				
					
0950:					
					
	sErrorDescription1 := 'Overload 2.  95% or more of max current command continued for 1 sec. or more.';				
	sErrorDescription2 := 'Check the load weight and the robot for collisions, etc';				
					
0960:					
					
	sErrorDescription1 := 'Excessive error 1.  The position error exceeded at servo ON.';				
	sErrorDescription2 := 'Check the load weight and press, etc';				
					
0970:					
					
	sErrorDescription1 := 'Excessive error 2.  The position error exceeded at servo OFF.';				
	sErrorDescription2 := 'Check the moving robot arm by something power';				
					
0980:					
					
	sErrorDescription1 := 'Excessive error 3.  Abnormal motor power line connection.';				
	sErrorDescription2 := 'Check the connection of motor power line';				
					
0990:					
					
	sErrorDescription1 := 'Collision detection 0.  A collision detection method 1 error was detected during the G0.';				
	sErrorDescription2 := 'Release the collision state';				
					
1000:					
					
	sErrorDescription1 := 'Collision detection 1.  A collision detection method 1 error was detected during the G1.';				
	sErrorDescription2 := 'Release the collision state';				
					
1010:					
					
	sErrorDescription1 := 'Collision detection.  Robot collided with something, or COLLVL is too low.';				
	sErrorDescription2 := 'Removal of the factor of a collision, or improve COLLVL';				
					
1020:					
					
	sErrorDescription1 := 'Servo AMP over-regeneration.  Overheating of the regenerative resistor was detected.';				
	sErrorDescription2 := 'Check the regeneration capacity and parameter SVPTYPE';				
					
1030:					
					
	sErrorDescription1 := 'Power supply over-regeneratio.  The power supplys regeneration capacity limit was exceeded.';				
	sErrorDescription2 := 'Wait at least 15min in the power ON state, and then turn OFF';				
					
1040:					
					
	sErrorDescription1 := 'Encoder init communication er.  Initial communication with the encoder was not possible.';				
	sErrorDescription2 := 'Check the encoder cable connection';				
					
1050:					
					
	sErrorDescription1 := ' Encoder init communication er.  Initial communication with the encoder was not possible.';				
	sErrorDescription2 := 'Check the encoder cable connection';				
					
1060:					
					
	sErrorDescription1 := ' Encoder communication error.  Communication between the encoder and detector was cut off.';				
	sErrorDescription2 := 'Check the encoder cable connection';				
					
1070:					
					
	sErrorDescription1 := 'Encoder communication error.  Communication between the encoder and detector was cut off.';				
	sErrorDescription2 := 'Check the encoder cable connection';				
					
1080:					
					
	sErrorDescription1 := 'Servo AMP communication error.  Communication from the RC was cut off.';				
	sErrorDescription2 := 'Check the communication cable connection and conductivity';				
					
1090:					
					
	sErrorDescription1 := 'Servo AMP initialization erro.  Initialization of the servo amplifier failed.';				
	sErrorDescription2 := 'Check the servo axis settings (parameters, rotary switches)';				
					
1100:					
					
	sErrorDescription1 := 'Servo com. receive error.  Abnormality occurred in data reception from a servo amplifier.';				
	sErrorDescription2 := 'Check the communication cable connection and conductivity';				
					
1110:					
					
	sErrorDescription1 := 'Servo com. receive error.  Abnormality occurred in data reception from a servo amplifier.';				
	sErrorDescription2 := 'Check the communication cable connection and conductivity';				
					
1120:					
					
	sErrorDescription1 := 'Encoder ABS position data los.  The absolute position data in the detector was lost.';				
	sErrorDescription2 := 'Check the battery voltage and detector cable';				
					
1130:					
					
	sErrorDescription1 := 'Encoder per rotation data err.  An error was detected in the encoders per rotation data.';				
	sErrorDescription2 := 'Check the repeatability and ambient environment';				
					
1140:					
					
	sErrorDescription1 := 'SRV-AMP Comm. data error (CRC.  A CRC error was detected in the data from the RC.';				
	sErrorDescription2 := 'Check the communication cable connection and conductivity';				
					
1150:					
					
	sErrorDescription1 := 'Large command position.  The command position from the RC is abnormally large.';				
	sErrorDescription2 := 'Check the communication cable connection and conductivity';				
					
1160:					
					
	sErrorDescription1 := 'SRV-AMP Comm. error (frame).  An error was detected in the communication frame from the RC.';				
	sErrorDescription2 := 'Check the communication cable connection and conductivity';				
					
1170:					
					
	sErrorDescription1 := 'SRV-AMP Comm. error (info).  Error in the communication information from the RC.';				
	sErrorDescription2 := 'Check the communication cable connection and conductivity';				
					
1180:					
					
	sErrorDescription1 := 'Servo amplifier feedback erro.  A pulse was skipped in the detector feedback signal.';				
	sErrorDescription2 := 'Check the encoder cable connection and conductivity';				
					
1190:					
					
	sErrorDescription1 := 'Servo amplifier feedback erro.  A deviation occurred in the motor end and machine end positions.';				
	sErrorDescription2 := 'Check the encoder';				
					
1200:					
					
	sErrorDescription1 := 'SRV-AMP Comm. data error (CRC.  CRC error in the communication data from the servo amplifier.';				
	sErrorDescription2 := 'Check the communication cable connection and conductivity';				
					
1210:					
					
	sErrorDescription1 := 'SRV-AMP Comm. data error (ID).  Data ID error in the communication data from the servo AMP.';				
	sErrorDescription2 := 'Check the communication cable connection and conductivity';				
					
1220:					
					
	sErrorDescription1 := 'SRV-AMP Comm. data error(axis.  Axis No error in the communication data from the servo AMP.';				
	sErrorDescription2 := 'Check the communication cable connection and conductivity';				
					
1230:					
					
	sErrorDescription1 := 'SRV-AMP Comm. data error(SubI.  Sub ID error in the communication data from the servo AMP.';				
	sErrorDescription2 := 'Check the communication cable connection and conductivity';				
					
1240:					
					
	sErrorDescription1 := 'SRV-AMP Comm. data error(fram.  No. of frames error in the communication data from servo AMP.';				
	sErrorDescription2 := 'Check the communication cable connection and conductivity';				
					
1250:					
					
	sErrorDescription1 := 'Servo amplifier parameter err.  An error was detected in the servo parameter.';				
	sErrorDescription2 := 'Change the servo parameter to an appropriate value';				
					
1360:					
					
	sErrorDescription1 := ' Absolute position counter err.  The counter of absolute position is illegal.';				
	sErrorDescription2 := 'Check the repeatability and ambient environment';				
					
1380:					
					
	sErrorDescription1 := ' Removing control axis (servo).  The axis removable command has been input from the controller.';				
	sErrorDescription2 := 'Reset the axis removable command';				
					
1390:					
					
	sErrorDescription1 := 'Emergency stop (Servo amplifi.  The emergency stop command has been input from the RC.';				
	sErrorDescription2 := 'Release the emergency stop state';				
					
1410:					
					
	sErrorDescription1 := 'Instantaneous power failure(S.  The power was momentarily interrupted.';				
	sErrorDescription2 := 'Check power spec., and wiring of power and external EMG. stop';				
					
1440:					
					
	sErrorDescription1 := 'System error (servo 1).  Trouble occurred in the current processing CPU.';				
	sErrorDescription2 := 'Turn the power OFF and ON';				
					
1450:					
					
	sErrorDescription1 := 'Instantaneous power interrupt.  The power was momentarily interrupted at the power supply.';				
	sErrorDescription2 := 'Check power spec., and wiring of power and external EMG. stop';				
					
1460:					
					
	sErrorDescription1 := 'Power supply overcurrent.  Overcurrent in the power module in the power supply.';				
	sErrorDescription2 := 'Check the AC power line, or change the power supply';				
					
1470:					
					
	sErrorDescription1 := 'Frequency error.  AC frequency is out of range.';				
	sErrorDescription2 := 'Check the AC power line frequency, or change the power supply';				
					
1480:					
					
	sErrorDescription1 := 'Power supply parameter error.  Illegal at the power supply parameter.';				
	sErrorDescription2 := 'Set the correct parameter';				
					
1490:					
					
	sErrorDescription1 := 'Power supply overheat.  Overheating of the power module or regenerative resistance.';				
	sErrorDescription2 := 'Check the fan on rear of power supply';				
					
1491:					
					
	sErrorDescription1 := ' Illegal converter thermal  se.  Overheating of  servo AMP converter..';				
	sErrorDescription2 := 'Turn the power OFF, wait a while, and then turn ON again.';				
					
1492:					
					
	sErrorDescription1 := ' Power supply converter overhe.  Overheating of the converter was detected.';				
	sErrorDescription2 := 'Turn the power OFF, wait a while, and then turn ON again';				
					
1493:					
					
	sErrorDescription1 := ' Rush resistance overheat.  Overheating of the rush resistance was detected.';				
	sErrorDescription2 := 'Turn the power OFF, wait a while, and then turn ON again';				
					
1494:					
					
	sErrorDescription1 := ' Discharge resistance overheat.  Overheating of the discharge resistance was detected.';				
	sErrorDescription2 := 'Turn the power OFF, wait a while, and then turn ON again';				
					
1500:					
					
	sErrorDescription1 := 'Motor combination error.  Illegal combination with additional servo amp and motor.';				
	sErrorDescription2 := 'Use additional servo amp with correctly combination';				
					
1510:					
					
	sErrorDescription1 := 'SRV-AMP USB comm. Error.  A communication error was detected between the servo amp and PC.';				
	sErrorDescription2 := 'Check the communication cable connection and conductivity';				
					
1530:					
					
	sErrorDescription1 := ' Encoder memory error.  .';				
	sErrorDescription2 := '';				
					
1540:					
					
	sErrorDescription1 := 'Communication error between u.  The transmission data between servo amplifier units is illegal.';				
	sErrorDescription2 := 'Check the communication cable connection and conductivity';				
					
1550:					
					
	sErrorDescription1 := 'Emergency stop is a breakdown.  The external emergency stop input is illegal.';				
	sErrorDescription2 := 'Turn the power OFF and ON once';				
					
1561:					
					
	sErrorDescription1 := 'Excessive error 4.  Axis moved during servo on process.';				
	sErrorDescription2 := 'It is necessary to change some parts when not improvement';				
					
1570:					
					
	sErrorDescription1 := 'Non-registered servo error.  A non-registered servo error occurred.';				
	sErrorDescription2 := 'If the warning cannot be reset, turn the power OFF and ON';				
					
1590:					
					
	sErrorDescription1 := ' System error (illegal EMG).  An non-registered emergency stop was input.';				
	sErrorDescription2 := '';				
					
1600:					
					
	sErrorDescription1 := 'System error (No robot setted.  None of the robots are set.';				
	sErrorDescription2 := 'Set the robots for at least one unit';				
					
1601:					
					
	sErrorDescription1 := ' Unmatched robot model.  Robot arm that connection is not correct.';				
	sErrorDescription2 := 'Please confirm the connected robot arm';				
					
1610:					
					
	sErrorDescription1 := 'System error (illegal MEMECH).  The setting parameter MEMECH is illegal.';				
	sErrorDescription2 := 'Set the correct MEMECH';				
					
1680:					
					
	sErrorDescription1 := 'Cannot servo ON (timeout).  The servo did not turn ON within the specified time.';				
	sErrorDescription2 := 'Check for errors in the servo amplifier';				
					
1681:					
					
	sErrorDescription1 := 'Unexpected servo OFF.  The servo turned OFF unexpectedly.';				
	sErrorDescription2 := 'Check for errors in the servo amplifier';				
					
1682:					
					
	sErrorDescription1 := ' Servo ON Timeout(Safety relay.  A main circuit voltage did not rise because of Safety relay.';				
	sErrorDescription2 := 'Check for errors in the Safety relay';				
					
1683:					
					
	sErrorDescription1 := ' Servo ON Timeout.(Contactor).  A main circuit voltage did not rise because of contactor welded..';				
	sErrorDescription2 := 'Check for errors in the contactor.';				
					
1790:					
					
	sErrorDescription1 := 'Illegal parameter (MEJAR).  The setting of parameter MEJAR is illegal.';				
	sErrorDescription2 := 'Correct the parameter MEJAR';				
					
1800:					
					
	sErrorDescription1 := 'Illegal parameter (MEMAR).  The setting of parameter MEMAR is illegal.';				
	sErrorDescription2 := 'Correct the parameter MEMAR';				
					
1810:					
					
	sErrorDescription1 := 'Illegal parameter (USERORG).  The setting of parameter USERORG is illegal.';				
	sErrorDescription2 := 'Correct the parameter USERORG';				
					
1861:					
					
	sErrorDescription1 := 'Illegal parameter (J1OFFSET).  The setting of parameter J1OFFSET is illegal.';				
	sErrorDescription2 := 'Correct the 2nd element of parameter J1OFFSET';				
					
1881:					
					
	sErrorDescription1 := 'Cooling fan stopped (add. axi.  Cooling fan of the add. axis amp. J1 might be out of order.';				
	sErrorDescription2 := 'Please exchange the cooling fan';				
					
1882:					
					
	sErrorDescription1 := 'Cooling fan stopped (add. axi.  Cooling fan of the add. axis amp. J2 might be out of order.';				
	sErrorDescription2 := 'Please exchange the cooling fan';				
					
1883:					
					
	sErrorDescription1 := 'Cooling fan stopped (add. axi.  Cooling fan of the add. axis amp. J3 might be out of order.';				
	sErrorDescription2 := 'Please exchange the cooling fan';				
					
1884:					
					
	sErrorDescription1 := 'Cooling fan stopped (add. axi.  Cooling fan of the add. axis amp. J4 might be out of order.';				
	sErrorDescription2 := 'Please exchange the cooling fan';				
					
1885:					
					
	sErrorDescription1 := 'Cooling fan stopped (add. axi.  Cooling fan of the add. axis amp. J5 might be out of order.';				
	sErrorDescription2 := 'Please exchange the cooling fan';				
					
1886:					
					
	sErrorDescription1 := 'Cooling fan stopped (add. axi.  Cooling fan of the add. axis amp. J6 might be out of order.';				
	sErrorDescription2 := 'Please exchange the cooling fan';				
					
1887:					
					
	sErrorDescription1 := 'Cooling fan stopped (add. axi.  Cooling fan of the add. axis amp. J7 might be out of order.';				
	sErrorDescription2 := 'Please exchange the cooling fan';				
					
1888:					
					
	sErrorDescription1 := 'Cooling fan stopped (add. axi.  Cooling fan of the add. axis amp. J8 might be out of order.';				
	sErrorDescription2 := 'Please exchange the cooling fan';				
					
1900:					
					
	sErrorDescription1 := 'Cooling fan stopped (pow. sup.  The power supply cooling fan stopped.';				
	sErrorDescription2 := 'Confirm the rotation of the power supply cooling fan';				
					
1950:					
					
	sErrorDescription1 := ' Additional axis AMP error.  Alarm of the additional axis servo amplifier was detected.';				
	sErrorDescription2 := 'Please refer to the manual of servo amplifier.';				
					
2031:					
					
	sErrorDescription1 := 'Illegal parameter(JOGTSJ,JOGJ.  Illegal parameter(JOGTSJ,JOGJSP).';				
	sErrorDescription2 := 'Set value under 5';				
					
2090:					
					
	sErrorDescription1 := 'In interference zone n.  Movement inside the user-defined area range was attempted.';				
	sErrorDescription2 := 'Adjust the position data';				
					
2111:					
					
	sErrorDescription1 := 'Free plane 1 overrun.  Movement outside the free plane 1 was attempted.';				
	sErrorDescription2 := 'Change the position data';				
					
2112:					
					
	sErrorDescription1 := 'Free plane 2 overrun.  Movement outside the free plane 2 was attempted.';				
	sErrorDescription2 := 'Change the position data';				
					
2113:					
					
	sErrorDescription1 := 'Free plane 3 overrun.  Movement outside the free plane 3 was attempted.';				
	sErrorDescription2 := 'Change the position data';				
					
2114:					
					
	sErrorDescription1 := 'Free plane 4 overrun.  Movement outside the free plane 4 was attempted.';				
	sErrorDescription2 := 'Change the position data';				
					
2115:					
					
	sErrorDescription1 := 'Free plane 5 overrun.  Movement outside the free plane 5 was attempted.';				
	sErrorDescription2 := 'Change the position data';				
					
2116:					
					
	sErrorDescription1 := 'Free plane 6 overrun.  Movement outside the free plane 6 was attempted.';				
	sErrorDescription2 := 'Change the position data';				
					
2117:					
					
	sErrorDescription1 := 'Free plane 7 overrun.  Movement outside the free plane 7 was attempted.';				
	sErrorDescription2 := 'Change the position data';				
					
2118:					
					
	sErrorDescription1 := 'Free plane 8 overrun.  Movement outside the free plane 8 was attempted.';				
	sErrorDescription2 := 'Change the position data';				
					
2119:					
					
	sErrorDescription1 := ' Free plane 9 overrun.  Movement outside the free plane 9 was attempted.';				
	sErrorDescription2 := 'Change the position data';				
					
2120:					
					
	sErrorDescription1 := ' Free plane 10 overrun.  Movement outside the free plane 10 was attempted.';				
	sErrorDescription2 := 'Change the position data';				
					
2121:					
					
	sErrorDescription1 := ' Free plane 11 overrun.  Movement outside the free plane 11 was attempted.';				
	sErrorDescription2 := 'Change the position data';				
					
2122:					
					
	sErrorDescription1 := ' Free plane 12 overrun.  Movement outside the free plane 12 was attempted.';				
	sErrorDescription2 := 'Change the position data';				
					
2123:					
					
	sErrorDescription1 := ' Free plane 13 overrun.  Movement outside the free plane 13 was attempted.';				
	sErrorDescription2 := 'Change the position data';				
					
2124:					
					
	sErrorDescription1 := ' Free plane 14 overrun.  Movement outside the free plane 14 was attempted.';				
	sErrorDescription2 := 'Change the position data';				
					
2125:					
					
	sErrorDescription1 := ' Free plane 15 overrun.  Movement outside the free plane 15 was attempted.';				
	sErrorDescription2 := 'Change the position data';				
					
2126:					
					
	sErrorDescription1 := ' Free plane 16 overrun.  Movement outside the free plane 16 was attempted.';				
	sErrorDescription2 := 'Change the position data';				
					
2129:					
					
	sErrorDescription1 := 'Free plane limit data illegal.  The free plane data setting value is illegal.';				
	sErrorDescription2 := 'Set the correct free plane setting data';				
					
2130:					
					
	sErrorDescription1 := 'Speed is excessive (command).  The axis speed limit was exceeded.';				
	sErrorDescription2 := 'Reduce the robot motion speed,insert an OVRD,ACCEL or SPD';				
					
2131:					
					
	sErrorDescription1 := 'J1 Speed is excessive (comman.  The axis J1 speed limit was exceeded.';				
	sErrorDescription2 := 'Reduce the robot motion speed,insert an OVRD,ACCEL or SPD';				
					
2132:					
					
	sErrorDescription1 := 'J2 Speed is excessive (comman.  The axis J2 speed limit was exceeded.';				
	sErrorDescription2 := 'Reduce the robot motion speed,insert an OVRD,ACCEL or SPD';				
					
2133:					
					
	sErrorDescription1 := 'J3 Speed is excessive (comman.  The axis J3 speed limit was exceeded.';				
	sErrorDescription2 := 'Reduce the robot motion speed,insert an OVRD,ACCEL or SPD';				
					
2134:					
					
	sErrorDescription1 := 'J4 Speed is excessive (comman.  The axis J4 speed limit was exceeded.';				
	sErrorDescription2 := 'Reduce the robot motion speed,insert an OVRD,ACCEL or SPD';				
					
2135:					
					
	sErrorDescription1 := 'J5 Speed is excessive (comman.  The axis J5 speed limit was exceeded.';				
	sErrorDescription2 := 'Reduce the robot motion speed,insert an OVRD,ACCEL or SPD';				
					
2136:					
					
	sErrorDescription1 := 'J6 Speed is excessive (comman.  The axis J6 speed limit was exceeded.';				
	sErrorDescription2 := 'Reduce the robot motion speed,insert an OVRD,ACCEL or SPD';				
					
2137:					
					
	sErrorDescription1 := 'J7 Speed is excessive (comman.  The axis J7 speed limit was exceeded.';				
	sErrorDescription2 := 'Reduce the robot motion speed,insert an OVRD,ACCEL or SPD';				
					
2138:					
					
	sErrorDescription1 := 'J8 Speed is excessive (comman.  The axis J8 speed limit was exceeded.';				
	sErrorDescription2 := 'Reduce the robot motion speed,insert an OVRD,ACCEL or SPD';				
					
2140:					
					
	sErrorDescription1 := 'ABS limit over.  ABS limit over.';				
	sErrorDescription2 := 'JOG operation with LS release operation';				
					
2141:					
					
	sErrorDescription1 := 'J1 +ABS limit over.  J1 +ABS limit over.';				
	sErrorDescription2 := 'JOG operation with LS release operation';				
					
2142:					
					
	sErrorDescription1 := 'J2 +ABS limit over.  J2 +ABS limit over.';				
	sErrorDescription2 := 'JOG operation with LS release operation';				
					
2143:					
					
	sErrorDescription1 := 'J3 +ABS limit over.  J3 +ABS limit over.';				
	sErrorDescription2 := 'JOG operation with LS release operation';				
					
2144:					
					
	sErrorDescription1 := 'J4 +ABS limit over.  J4 +ABS limit over.';				
	sErrorDescription2 := 'JOG operation with LS release operation';				
					
2145:					
					
	sErrorDescription1 := 'J5 +ABS limit over.  J5 +ABS limit over.';				
	sErrorDescription2 := 'JOG operation with LS release operation';				
					
2146:					
					
	sErrorDescription1 := 'J6 +ABS limit over.  J6 +ABS limit over.';				
	sErrorDescription2 := 'JOG operation with LS release operation';				
					
2147:					
					
	sErrorDescription1 := 'J7 +ABS limit over.  J7 +ABS limit over.';				
	sErrorDescription2 := 'JOG operation with LS release operation';				
					
2148:					
					
	sErrorDescription1 := 'J8 +ABS limit over.  J8 +ABS limit over.';				
	sErrorDescription2 := 'JOG operation with LS release operation';				
					
2151:					
					
	sErrorDescription1 := 'J1 -ABS limit over.  J1 -ABS limit over.';				
	sErrorDescription2 := 'JOG operation with LS release operation';				
					
2152:					
					
	sErrorDescription1 := 'J2 -ABS limit over.  J2 -ABS limit over.';				
	sErrorDescription2 := 'JOG operation with LS release operation';				
					
2153:					
					
	sErrorDescription1 := 'J3 -ABS limit over.  J3 -ABS limit over.';				
	sErrorDescription2 := 'JOG operation with LS release operation';				
					
2154:					
					
	sErrorDescription1 := 'J4 -ABS limit over.  J4 -ABS limit over.';				
	sErrorDescription2 := 'JOG operation with LS release operation';				
					
2155:					
					
	sErrorDescription1 := 'J5 -ABS limit over.  J5 -ABS limit over.';				
	sErrorDescription2 := 'JOG operation with LS release operation';				
					
2156:					
					
	sErrorDescription1 := 'J6 -ABS limit over.  J6 -ABS limit over.';				
	sErrorDescription2 := 'JOG operation with LS release operation';				
					
2157:					
					
	sErrorDescription1 := 'J7 -ABS limit over.  J7 -ABS limit over.';				
	sErrorDescription2 := 'JOG operation with LS release operation';				
					
2158:					
					
	sErrorDescription1 := 'J8 -ABS limit over.  J8 -ABS limit over.';				
	sErrorDescription2 := 'JOG operation with LS release operation';				
					
2160:					
					
	sErrorDescription1 := 'Joint angle exceeds the limit.  Joint angle exceeds the limit.';				
	sErrorDescription2 := 'Change the position data';				
					
2161:					
					
	sErrorDescription1 := 'J1 (+) angle exceeds the limi.  J1(+) angle exceeds the limit.';				
	sErrorDescription2 := 'Change the position data';				
					
2162:					
					
	sErrorDescription1 := 'J2 (+) angle exceeds the limi.  J2(+) angle exceeds the limit.';				
	sErrorDescription2 := 'Change the position data';				
					
2163:					
					
	sErrorDescription1 := 'J3 (+) angle exceeds the limi.  J3(+) angle exceeds the limit.';				
	sErrorDescription2 := 'Change the position data';				
					
2164:					
					
	sErrorDescription1 := 'J4 (+) angle exceeds the limi.  J4(+) angle exceeds the limit.';				
	sErrorDescription2 := 'Change the position data';				
					
2165:					
					
	sErrorDescription1 := 'J5 (+) angle exceeds the limi.  J5(+) angle exceeds the limit.';				
	sErrorDescription2 := 'Change the position data';				
					
2166:					
					
	sErrorDescription1 := 'J6 (+) angle exceeds the limi.  J6(+) angle exceeds the limit.';				
	sErrorDescription2 := 'Change the position data';				
					
2167:					
					
	sErrorDescription1 := 'J7 (+) angle exceeds the limi.  J7(+) angle exceeds the limit.';				
	sErrorDescription2 := 'Change the position data';				
					
2168:					
					
	sErrorDescription1 := 'J8 (+) angle exceeds the limi.  J8(+) angle exceeds the limit.';				
	sErrorDescription2 := 'Change the position data';				
					
2171:					
					
	sErrorDescription1 := 'J1 (-) angle exceeds the limi.  J1(-) angle exceeds the limit.';				
	sErrorDescription2 := 'Change the position data';				
					
2172:					
					
	sErrorDescription1 := 'J2 (-) angle exceeds the limi.  J2(-) angle exceeds the limit.';				
	sErrorDescription2 := 'Change the position data';				
					
2173:					
					
	sErrorDescription1 := 'J3 (-) angle exceeds the limi.  J3(-) angle exceeds the limit.';				
	sErrorDescription2 := 'Change the position data';				
					
2174:					
					
	sErrorDescription1 := 'J4 (-) angle exceeds the limi.  J4(-) angle exceeds the limit.';				
	sErrorDescription2 := 'Change the position data';				
					
2175:					
					
	sErrorDescription1 := 'J5 (-) angle exceeds the limi.  J5(-) angle exceeds the limit.';				
	sErrorDescription2 := 'Change the position data';				
					
2176:					
					
	sErrorDescription1 := 'J6 (-) angle exceeds the limi.  J6(-) angle exceeds the limit.';				
	sErrorDescription2 := 'Change the position data';				
					
2177:					
					
	sErrorDescription1 := 'J7 (-) angle exceeds the limi.  J7(-) angle exceeds the limit.';				
	sErrorDescription2 := 'Change the position data';				
					
2178:					
					
	sErrorDescription1 := 'J8 (-) angle exceeds the limi.  J8(-) angle exceeds the limit.';				
	sErrorDescription2 := 'Change the position data';				
					
2180:					
					
	sErrorDescription1 := 'X,Y,Z data exceeds the limit.  X,Y,Z data exceeds the limit.';				
	sErrorDescription2 := 'Change the position data';				
					
2181:					
					
	sErrorDescription1 := 'X(+) data exceeds the limit.  X(+) data exceeds the limit.';				
	sErrorDescription2 := 'Change the position data';				
					
2182:					
					
	sErrorDescription1 := 'Y(+) data exceeds the limit.  Y(+) data exceeds the limit.';				
	sErrorDescription2 := 'Change the position data';				
					
2183:					
					
	sErrorDescription1 := 'Z(+) data exceeds the limit.  Z(+) data exceeds the limit.';				
	sErrorDescription2 := 'Change the position data';				
					
2191:					
					
	sErrorDescription1 := 'X(-) data exceeds the limit.  X(-) data exceeds the limit.';				
	sErrorDescription2 := 'Change the position data';				
					
2192:					
					
	sErrorDescription1 := 'Y(-) data exceeds the limit.  Y(-) data exceeds the limit.';				
	sErrorDescription2 := 'Change the position data';				
					
2193:					
					
	sErrorDescription1 := 'Z(-) data exceeds the limit.  Z(-) data exceeds the limit.';				
	sErrorDescription2 := 'Change the position data';				
					
2200:					
					
	sErrorDescription1 := ' SLP (ROBOT position error).  Safety Position monitoring detected over the position limits.';				
	sErrorDescription2 := 'Please confirm the robot movement or related parameter setting';				
					
2210:					
					
	sErrorDescription1 := ' STR (ROBOT torque error).  Safety Torque Range monitoring detected over the torque thresh..';				
	sErrorDescription2 := 'Please confirm the robot movement or related parameter setting';				
					
2220:					
					
	sErrorDescription1 := ' Mismatch of Dual Safety Input.  State of the redundant wiring do not match (Dual Safty Input).';				
	sErrorDescription2 := 'Please check the wiring or parameter';				
					
2230:					
					
	sErrorDescription1 := ' Mismatch of Dual Safety Outpu.  State of the redundant wiring do not match (Dual Safty Output).';				
	sErrorDescription2 := 'If this error recurs, please contact us';				
					
2231:					
					
	sErrorDescription1 := ' Mismatch of Dual Safety Outpu.  State of Dual Safty Output and the feedback do not match.';				
	sErrorDescription2 := 'If this error recurs, please contact us';				
					
2240:					
					
	sErrorDescription1 := ' Origin data was changed.  Origin data was changed under the position monitor processing.';				
	sErrorDescription2 := 'Turn the power OFF and ON once';				
					
2260:					
					
	sErrorDescription1 := ' Safety function is not execut.  Extended safety unit of the robot safety option is not installed.';				
	sErrorDescription2 := 'Please install the extended safety unit';				
					
2261:					
					
	sErrorDescription1 := ' Extended safety units No. er.  The extended safety unit’s station No. is illegal.';				
	sErrorDescription2 := 'Set the extended safety unit’s station No. to 2';				
					
2280:					
					
	sErrorDescription1 := ' SS1 deceleration time exceede.  The robot did not stop within deceleration time from SS1 enabled.';				
	sErrorDescription2 := 'Please confirm the robot movement or related parameter setting';				
					
2281:					
					
	sErrorDescription1 := ' SS2 deceleration time exceede.  The robot did not stop within deceleration time from SS2 enabled.';				
	sErrorDescription2 := 'Please confirm the robot movement or related parameter setting';				
					
2282:					
					
	sErrorDescription1 := ' SOS error.  Detect the change of position FB on SOS.';				
	sErrorDescription2 := 'Please check external force or related parameter settings';				
					
2300:					
					
	sErrorDescription1 := ' SLS (Joint Speed Error).  Speed monitor detected the speed over.';				
	sErrorDescription2 := 'Please confirm the robot movement or related parameter setting';				
					
2310:					
					
	sErrorDescription1 := ' SLS (XYZ Speed Error).  Speed monitor detected the speed over.';				
	sErrorDescription2 := 'Please confirm the robot movement or related parameter setting';				
					
2320:					
					
	sErrorDescription1 := ' SF (Robot control error).  Command position and F/B position are not corresponding.';				
	sErrorDescription2 := 'Please confirm the robot movement and presence of interference';				
					
2330:					
					
	sErrorDescription1 := ' SF (Servo control error).  Abnormality of Servo Control was detected.';				
	sErrorDescription2 := 'Please confirm the robot movement and presence of interference';				
					
2340:					
					
	sErrorDescription1 := ' SF (Motion command error).  Abnormality of Command Position was detected.';				
	sErrorDescription2 := 'Turn the power OFF and ON once';				
					
2350:					
					
	sErrorDescription1 := ' SLS (Motor drive command erro.  Speed monitor (Servo) detected the position command speed excess.';				
	sErrorDescription2 := 'Turn the power OFF and ON once';				
					
2360:					
					
	sErrorDescription1 := ' SF (Encoder data error).  Abnormality of Encoder Data was detected.';				
	sErrorDescription2 := 'Turn the power OFF and ON once';				
					
2370:					
					
	sErrorDescription1 := ' SF (Process error).  The Safety Function is not normally executed.';				
	sErrorDescription2 := 'Turn the power OFF and ON once';				
					
2380:					
					
	sErrorDescription1 := ' SF (SCPU Process error).  Abnormality of the Safety Function was detected.';				
	sErrorDescription2 := 'Turn the power OFF and ON once';				
					
2420:					
					
	sErrorDescription1 := ' Collision avoidance comm. err.  Collision avoidance comm. error.';				
	sErrorDescription2 := 'Check the robot controller';				
					
2500:					
					
	sErrorDescription1 := 'Tracking encoder data error.  An error was detected in the tracking encoder data.';				
	sErrorDescription2 := 'Check the repeatability and ambient environment';				
					
2570:					
					
	sErrorDescription1 := ' Installation slot error..  Q173DPX is installed in slot 0-2 of a basic base..';				
	sErrorDescription2 := 'Install Q173DPX to slot 3-11.';				
					
2630:					
					
	sErrorDescription1 := ' Setting the value of DISPCTYP.  Out of range value is set to DISPCTYP.';				
	sErrorDescription2 := 'Please confirm the value of DISPCTYP';				
					
2640:					
					
	sErrorDescription1 := ' Add axis FLS signal is input.  Add axis FLS signal is input.';				
	sErrorDescription2 := 'JOG operation with LS release operation';				
					
2650:					
					
	sErrorDescription1 := ' Add axis RLS signal is input.  Add axis RLS signal is input.';				
	sErrorDescription2 := 'JOG operation with LS release operation';				
					
2663:					
					
	sErrorDescription1 := ' Origin data was changed.  Origin data was changed about the base cooperation target axis.';				
	sErrorDescription2 := 'Turn the power OFF and ON once';				
					
2760:					
					
	sErrorDescription1 := ' Correction limit (F.Ctrl).  The correction value of the force control exceeded the limit.';				
	sErrorDescription2 := 'Please confirm the movement of the robot';				
					
2770:					
					
	sErrorDescription1 := ' exceeds the joint limit.  Position of force control exceeds the joint limit.';				
	sErrorDescription2 := 'Please revice the position';				
					
2780:					
					
	sErrorDescription1 := ' exceeds the speed limit.  Position of force control exceeds the speed limit.';				
	sErrorDescription2 := 'Please revice the operation';				
					
2820:					
					
	sErrorDescription1 := 'Illegal ACCEL ratio.  Illegal ACCEL ratio.';				
	sErrorDescription2 := 'Set the correct ACCEL ratio';				
					
2840:					
					
	sErrorDescription1 := 'System error (ipol parameters.  Parameters setting is illegal.';				
	sErrorDescription2 := 'Set the correct parameters';				
					
2850:					
					
	sErrorDescription1 := 'System error (ipol norm).  System error (ipol norm).';				
	sErrorDescription2 := 'Please call S.C.';				
					
2860:					
					
	sErrorDescription1 := 'System error (ipol type).  Illegal interpolation type.';				
	sErrorDescription2 := 'Please call S.C.';				
					
2870:					
					
	sErrorDescription1 := 'System error(ipol data undef).  Ipol data is undefined.';				
	sErrorDescription2 := 'Please call S.C.';				
					
2880:					
					
	sErrorDescription1 := 'System error (ipol data area).  No more ipol data area.';				
	sErrorDescription2 := 'Please call S.C.';				
					
2890:					
					
	sErrorDescription1 := 'System error (undefined err).  System error (undefined err).';				
	sErrorDescription2 := 'Please call S.C.';				
					
3983:					
					
	sErrorDescription1 := 'Cannot execute CNT movement.  A structural flag or the angle of the joint is not corresponding.';				
	sErrorDescription2 := 'It surely positions it by DLY command etc';				
					
3985:					
					
	sErrorDescription1 := 'Cannot be passsed (singularit.  Robot passes position which is very near the singular point.';				
	sErrorDescription2 := 'Adjust the teaching position';				
					
3988:					
					
	sErrorDescription1 := ' Cannot calculate the position.  Position of force control could not convert a joint angle.';				
	sErrorDescription2 := 'Please revice the position';				
					
5000:					
					
	sErrorDescription1 := 'TB Enable key is ON.  The TB Enable key was ON in the AUTO mode.';				
	sErrorDescription2 := 'OFF the TB Enable key, or enter the TEACH mode';				
					
6000:					
					
	sErrorDescription1 := ' Please execute the all backup.  New error log information was made..';				
	sErrorDescription2 := 'You can reset the error,if "SPCERR" input is ON (Rising edge).';				
					
6100:					
					
	sErrorDescription1 := ' The module is not installed.  The module for the Network Base card is not installed.';				
	sErrorDescription2 := 'Please install the module for the Network Base card';				
					
6101:					
					
	sErrorDescription1 := ' Unsupported module is install.  Unsupported module is installed in the Network Base card.';				
	sErrorDescription2 := 'Please exchange the module';				
					
6110:					
					
	sErrorDescription1 := ' More TZ535 cards are installe.  Only one TZ535 card can be installed.';				
	sErrorDescription2 := 'Please install only one TZ535 card';				
					
6111:					
					
	sErrorDescription1 := ' Other field cards are install.  Only one fieldbus card can be installed.';				
	sErrorDescription2 := 'Only one fieldbus card is installed';				
					
6120:					
					
	sErrorDescription1 := ' Network Base card failure.  Abnormality of the Network Base card is detected.';				
	sErrorDescription2 := 'Please exchange the Network Base card';				
					
6140:					
					
	sErrorDescription1 := ' Parameter error.  Parameter setting is illegal.';				
	sErrorDescription2 := 'Please check the parameter setting';				
					
6510:					
					
	sErrorDescription1 := 'RS232C Parameter illgal.  Setup the parameter.';				
	sErrorDescription2 := 'Setup parameter and the power OFF';				
					
6520:					
					
	sErrorDescription1 := 'RS422 Parameter illgal.  Setup the parameter.';				
	sErrorDescription2 := 'Setup parameter and the power OFF';				
					
6530:					
					
	sErrorDescription1 := 'COMDEV parameter is illegal.  COMDEV parameter is illegal.';				
	sErrorDescription2 := 'Correct COMDEV parameter';				
					
6640:					
					
	sErrorDescription1 := 'Illegal param (special signal.  The parameter setting is illegal.';				
	sErrorDescription2 := 'Correct the parameter';				
					
6680:					
					
	sErrorDescription1 := ' Mismatch of Safety Input.  State of the redundant wiring do not match.(Safety Input).';				
	sErrorDescription2 := 'Please check the wiring or parameter';				
					
6681:					
					
	sErrorDescription1 := ' Mismatch of Safety Input1.  State of the redundant wiring do not match.(Safety Input 1).';				
	sErrorDescription2 := 'Please check the wiring or parameter';				
					
6682:					
					
	sErrorDescription1 := ' Mismatch of Safety Input2.  State of the redundant wiring do not match.(Safety Input 2).';				
	sErrorDescription2 := 'Please check the wiring or parameter';				
					
6683:					
					
	sErrorDescription1 := ' Mismatch of Safety Input3.  State of the redundant wiring do not match.(Safety Input 3).';				
	sErrorDescription2 := 'Please check the wiring or parameter';				
					
6690:					
					
	sErrorDescription1 := ' Safety Input Process error.  Abnormality of the Safety Input was detected.';				
	sErrorDescription2 := 'Turn the power OFF and ON once';				
					
7030:					
					
	sErrorDescription1 := 'System error (param size over.  Parameter file size over.';				
	sErrorDescription2 := 'Contact the maker';				
					
7050:					
					
	sErrorDescription1 := 'File is illegal.  The file is illegal.';				
	sErrorDescription2 := 'Do not use this file';				
					
7060:					
					
	sErrorDescription1 := 'System error (RAM area full).  System RAM area is full.';				
	sErrorDescription2 := 'Contact the maker';				
					
7100:					
					
	sErrorDescription1 := ' Robot arm serial number misma.  Robot arm that connection was replaced.';				
	sErrorDescription2 := 'Execute restoration of preventive maintenance data, or reset';				
					
7101:					
					
	sErrorDescription1 := ' Backup serial number mismatch.  Robot arm and backup data are the different serial number.';				
	sErrorDescription2 := 'Please use the backup data matching robot arm';				
					
7102:					
					
	sErrorDescription1 := ' Backup file version is differ.  Preventive maintenance function backup file version mismatch.';				
	sErrorDescription2 := 'Please select the backup file of the corresponding version';				
					
7300:					
					
	sErrorDescription1 := 'Loading the parameter file..  Turn the power OFF and ON once.';				
	sErrorDescription2 := 'Turn the power OFF and ON once';				
					
7600:					
					
	sErrorDescription1 := ' Illegal parameter (AXMENO).  The additional axis robot No. is incorrect.';				
	sErrorDescription2 := 'Correct parameter AXMENO,AXUNUM';				
					
7601:					
					
	sErrorDescription1 := ' Illegal parameter (AXJNO).  The additional axis No. is illegal.';				
	sErrorDescription2 := 'Correct parameter AXMENO';				
					
7602:					
					
	sErrorDescription1 := ' Duplicate parameter (AXJNO).  The additional axis No. has been used in duplicate.';				
	sErrorDescription2 := 'Correct parameter AXMENO';				
					
7603:					
					
	sErrorDescription1 := ' Illegal parameter (AXUNT).  The additional axis unit is incorrect.';				
	sErrorDescription2 := 'Correct parameter AXMUNT';				
					
7604:					
					
	sErrorDescription1 := ' Illegal parameter (AXACC).  The additional axis acceleration time is incorrect.';				
	sErrorDescription2 := 'Correct parameter AXACC';				
					
7605:					
					
	sErrorDescription1 := ' Illegal parameter (AXDCC).  The additional axis deceleration time is incorrect.';				
	sErrorDescription2 := 'Correct parameter AXDCC';				
					
7606:					
					
	sErrorDescription1 := ' Illegal parameter (AXGRTN).  The additional axis gear ratio denominator is incorrect.';				
	sErrorDescription2 := 'Correct parameter AXGRTN';				
					
7607:					
					
	sErrorDescription1 := ' Illegal parameter (AXGRTD).  The additional axis gear ratio numerator is incorrect.';				
	sErrorDescription2 := 'Correct parameter AXGRTD';				
					
7608:					
					
	sErrorDescription1 := ' Illegal parameter (AXMOTSET).  The additional axis motor setting validity flag is incorrect.';				
	sErrorDescription2 := 'Correct parameter AXMOTSET';				
					
7609:					
					
	sErrorDescription1 := ' Illegal parameter (AXMREV).  The additional axis motor rated speed is incorrect.';				
	sErrorDescription2 := 'Correct parameter AXMREV';				
					
7610:					
					
	sErrorDescription1 := ' Illegal parameter (AXJMX).  The additional axis motor limit speed is incorrect.';				
	sErrorDescription2 := 'Correct parameter AXJMX';				
					
7611:					
					
	sErrorDescription1 := ' Illegal parameter (AXENCR).  The additional axis No. of encoder pulses is incorrect.';				
	sErrorDescription2 := 'Correct parameter AXENCR';				
					
7612:					
					
	sErrorDescription1 := ' Illegal parameter (AXJOGTS).  The additional axis JOG time constant is incorrect.';				
	sErrorDescription2 := 'Correct parameter AXJOGTS';				
					
7613:					
					
	sErrorDescription1 := ' Turn the power OFF and ON onc.  Turn the power OFF and ON once.';				
	sErrorDescription2 := 'Turn the power OFF and ON once';				
					
7620:					
					
	sErrorDescription1 := ' Plural Add-Axis cards are set.  This card can install one.';				
	sErrorDescription2 := 'Reinstall one card';				
					
7650:					
					
	sErrorDescription1 := ' Number of force sensors is wr.  Two or more force sensors are set to one robot.';				
	sErrorDescription2 := 'Please confirm the setting of parameter AXJNO and AXMENO';				
					
7651:					
					
	sErrorDescription1 := ' I/F unit initialization error.  Initialization of the force control I/F unit failed.';				
	sErrorDescription2 := 'Please confirm the connection and the power supply of I/F unit';				
					
7652:					
					
	sErrorDescription1 := ' I/F unit revision is illegal.  It does not correspond to revision of this force sensor I/F unit.';				
	sErrorDescription2 := 'Please contact the maker';				
					
7660:					
					
	sErrorDescription1 := ' Force sensor error.  The data of force sensor that exceeded the limitation.';				
	sErrorDescription2 := 'Please confirm use and the state of force sensor';				
					
7700:					
					
	sErrorDescription1 := ' CC-Link card is illegal.  The master station is set.';				
	sErrorDescription2 := 'Please exchange the CC-Link card';				
					
7710:					
					
	sErrorDescription1 := ' Can not set the Master Station.  The master station is set..';				
	sErrorDescription2 := 'Set the station number except 0';				
					
7720:					
					
	sErrorDescription1 := ' Plural CC-Link cards are set.  CC-Link card can install one.';				
	sErrorDescription2 := 'Install only one CC-Link card';				
					
7760:					
					
	sErrorDescription1 := ' CC-Link initialization error.  Confirm the CC-Link error code.';				
	sErrorDescription2 := 'Confirm the CC-Link error code';				
					
7799:					
					
	sErrorDescription1 := ' CC-Link System error.  .';				
	sErrorDescription2 := '';				
					
7800:					
					
	sErrorDescription1 := ' Ethernet card initialization .  The Ethernet card is broken.';				
	sErrorDescription2 := 'Check the Ethernet board';				
					
7802:					
					
	sErrorDescription1 := ' Ethernet card is set in SLOT2.  Ethernet card is set in SLOT2 or 3.';				
	sErrorDescription2 := 'Install Ethernet card in SLOT1';				
					
7803:					
					
	sErrorDescription1 := ' Plural Ethernet cards are set.  Ethernet card can install one.';				
	sErrorDescription2 := 'Install the Ethernet card only in SLOT1';				
					
7810:					
					
	sErrorDescription1 := ' Ethernet parameter ERR.  Illegal parameter.';				
	sErrorDescription2 := 'Correct parameter';				
					
7820:					
					
	sErrorDescription1 := 'MXT/MXScommand timeout.  time over MXTTOUT parameter.';				
	sErrorDescription2 := 'Chech parameter MXTTOUT';				
					
7830:					
					
	sErrorDescription1 := 'Ethernet card is not installe.  Ethernet card is not installed, or command disable.';				
	sErrorDescription2 := 'Install Ethenet card';				
					
7840:					
					
	sErrorDescription1 := 'MXT/MXS command Illegal recei.  ・Illegal received data Illegal command position data (NAN/NUMBER) Different data type.';				
	sErrorDescription2 := 'Check MXT/MXS command and transmitted data Check transmitted command position data Check MXT/MXS command and transmitted data';				
					
7860:					
					
	sErrorDescription1 := ' SLMP error.  An error related to SLMP has occurred. .';				
	sErrorDescription2 := 'Please confirm the content by a detailed number of the error.';				
					
7861:					
					
	sErrorDescription1 := ' SLMP parameter error.  Illegal parameter. .';				
	sErrorDescription2 := 'Correct parameter. ';				
					
7870:					
					
	sErrorDescription1 := ' CC-Link IEF Basic Comm. Error.  Failure in the CC-Link IEF Commuication..';				
	sErrorDescription2 := 'Check the wiring and parameter setting on the master station.';				
					
7901:					
					
	sErrorDescription1 := ' OPTION1#1 Parameter illegal.  Setup the parameter.';				
	sErrorDescription2 := 'Setup patrameter and the power OFF';				
					
7902:					
					
	sErrorDescription1 := ' OPTION1#2 Parameter illegal.  Setup the parameter.';				
	sErrorDescription2 := 'Setup patrameter and the power OFF';				
					
7903:					
					
	sErrorDescription1 := ' OPTION1#3 Parameter illegal.  Setup the parameter.';				
	sErrorDescription2 := 'Setup patrameter and the power OFF';				
					
7911:					
					
	sErrorDescription1 := ' OPTION2#1 Parameter illegal.  Setup the parameter.';				
	sErrorDescription2 := 'Setup patrameter and the power OFF';				
					
7912:					
					
	sErrorDescription1 := ' OPTION2#2 Parameter illegal.  Setup the parameter.';				
	sErrorDescription2 := 'Setup patrameter and the power OFF';				
					
7913:					
					
	sErrorDescription1 := ' OPTION2#3 Parameter illegal.  Setup the parameter.';				
	sErrorDescription2 := 'Setup patrameter and the power OFF';				
					
7920:					
					
	sErrorDescription1 := ' Three EX-SIO I/F are installe.  Reinstall one or two cards to SLOT1 or 2.';				
	sErrorDescription2 := 'Remove the Expansion Serial card in SLOT3';				
					
7930:					
					
	sErrorDescription1 := ' EX-SIO card is set in SLOT3.  EX-SIO card is set in SLOT3.';				
	sErrorDescription2 := 'Remove the Expansion Serial card in SLOT 3';				
					
7990:					
					
	sErrorDescription1 := ' OptionCard illegal insert.  Check SLOT number.';				
	sErrorDescription2 := 'Power off, change the SLOT number';				
					
8000:					
					
	sErrorDescription1 := ' .  .';				
	sErrorDescription2 := '';				
					
8001:					
					
	sErrorDescription1 := ' .  .';				
	sErrorDescription2 := '';				
					
8002:					
					
	sErrorDescription1 := ' .  .';				
	sErrorDescription2 := '';				
					
8003:					
					
	sErrorDescription1 := ' .  .';				
	sErrorDescription2 := '';				
					
8004:					
					
	sErrorDescription1 := ' .  .';				
	sErrorDescription2 := '';				
					
8005:					
					
	sErrorDescription1 := ' .  .';				
	sErrorDescription2 := '';				
					
8010:					
					
	sErrorDescription1 := ' .  .';				
	sErrorDescription2 := '';				
					
8011:					
					
	sErrorDescription1 := ' .  .';				
	sErrorDescription2 := '';				
					
8012:					
					
	sErrorDescription1 := ' .  .';				
	sErrorDescription2 := '';				
					
8013:					
					
	sErrorDescription1 := ' .  .';				
	sErrorDescription2 := '';				
					
8014:					
					
	sErrorDescription1 := ' .  .';				
	sErrorDescription2 := '';				
					
8015:					
					
	sErrorDescription1 := ' Plural Vision cards are insta.  Vision card can be installed one.';				
	sErrorDescription2 := 'Reinstall one card';				
					
8016:					
					
	sErrorDescription1 := ' .  .';				
	sErrorDescription2 := '';				
					
8020:					
					
	sErrorDescription1 := ' .  .';				
	sErrorDescription2 := '';				
					
8021:					
					
	sErrorDescription1 := ' .  .';				
	sErrorDescription2 := '';				
					
8022:					
					
	sErrorDescription1 := ' .  .';				
	sErrorDescription2 := '';				
					
8023:					
					
	sErrorDescription1 := ' .  .';				
	sErrorDescription2 := '';				
					
8024:					
					
	sErrorDescription1 := ' .  .';				
	sErrorDescription2 := '';				
					
8025:					
					
	sErrorDescription1 := ' .  .';				
	sErrorDescription2 := '';				
					
8026:					
					
	sErrorDescription1 := ' .  .';				
	sErrorDescription2 := '';				
					
8027:					
					
	sErrorDescription1 := ' .  .';				
	sErrorDescription2 := '';				
					
8028:					
					
	sErrorDescription1 := ' .  .';				
	sErrorDescription2 := '';				
					
8029:					
					
	sErrorDescription1 := ' .  .';				
	sErrorDescription2 := '';				
					
8030:					
					
	sErrorDescription1 := ' .  .';				
	sErrorDescription2 := '';				
					
8031:					
					
	sErrorDescription1 := ' .  .';				
	sErrorDescription2 := '';				
					
8032:					
					
	sErrorDescription1 := ' .  .';				
	sErrorDescription2 := '';				
					
8033:					
					
	sErrorDescription1 := ' .  .';				
	sErrorDescription2 := '';				
					
8034:					
					
	sErrorDescription1 := ' .  .';				
	sErrorDescription2 := '';				
					
8035:					
					
	sErrorDescription1 := ' .  .';				
	sErrorDescription2 := '';				
					
8036:					
					
	sErrorDescription1 := ' .  .';				
	sErrorDescription2 := '';				
					
8037:					
					
	sErrorDescription1 := ' .  .';				
	sErrorDescription2 := '';				
					
8038:					
					
	sErrorDescription1 := ' .  .';				
	sErrorDescription2 := '';				
					
8039:					
					
	sErrorDescription1 := ' .  .';				
	sErrorDescription2 := '';				
					
8040:					
					
	sErrorDescription1 := ' .  .';				
	sErrorDescription2 := '';				
					
8130:					
					
	sErrorDescription1 := ' Multi-Hand Comm.error(RemoteI.  Communication line is illegal.';				
	sErrorDescription2 := 'Check the cable or power supply';				
					
8140:					
					
	sErrorDescription1 := ' Electric hand1 Comm.error(RIO.  Communication line is illegal.';				
	sErrorDescription2 := 'Check the cable or power supply';				
					
8150:					
					
	sErrorDescription1 := ' Electric hand2 Comm.error(RIO.  Communication line is illegal.';				
	sErrorDescription2 := 'Check the cable or power supply';				
					
8160:					
					
	sErrorDescription1 := ' Electric hand3 Comm.error(RIO.  Communication line is illegal.';				
	sErrorDescription2 := 'Check the cable or power supply';				
					
8201:					
					
	sErrorDescription1 := ' Illegal param (TPTMMG).  TPTMMG param is illegal.';				
	sErrorDescription2 := 'Correct TPTMMG parameter';				
					
8202:					
					
	sErrorDescription1 := ' Illegal param (TPERRNO).  TPERRNO param is illegal.';				
	sErrorDescription2 := 'Correct TPERRNO parameter';				
					
8203:					
					
	sErrorDescription1 := ' Illegal param (TPSIGNO).  TPSIGNO param is illegal.';				
	sErrorDescription2 := 'Correct TPSIGNO parameter';				
					
8204:					
					
	sErrorDescription1 := ' Illegal param (TRAP).  TRAP param is illegal.';				
	sErrorDescription2 := 'Correct TRAP parameter';				
					
8206:					
					
	sErrorDescription1 := ' failed in initialization (tra.  Turn the power OFF and power ON once.';				
	sErrorDescription2 := 'Please check communication state, setting, and command argument';				
					
8207:					
					
	sErrorDescription1 := ' failed in writing the data(tr.  failed in writing the data .';				
	sErrorDescription2 := 'Please do the operation over again';				
					
8320:					
					
	sErrorDescription1 := 'System Error (GETPOS).  Internal data of GETPOS is illegal.';				
	sErrorDescription2 := 'Turn the power OFF and ON once';				
					
8400:					
					
